KUKA KRL program: MyProgram_185().src

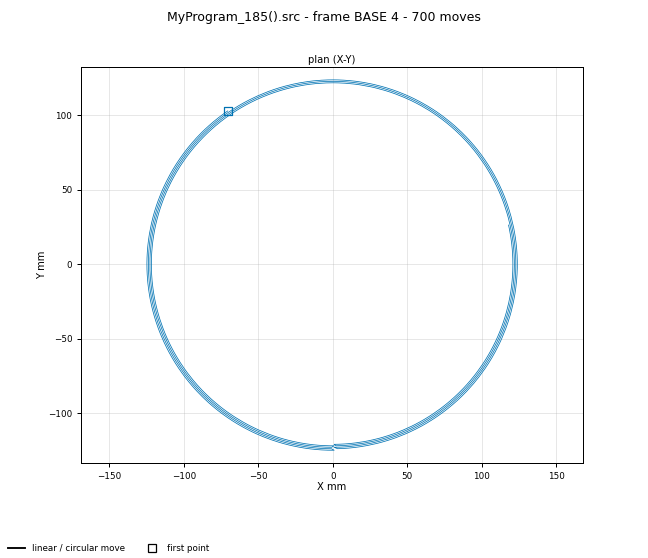
[picture p0: tool path of MyProgram_185().src in frame BASE 4, 700 of 700 moves have a stored position in this frame; points joined in program order, loops and branches not executed]
&ACCESS RVP
&REL 1
&PARAM TEMPLATE = C:\KRC\Roboter\Template\vorgabe
&PARAM EDITMASK = *
DEF MyProgram_185()
; ---- Setting reference (Base) ----
$BASE = BASE_DATA[4]

; --------------------------
; ---- Setting tool (TCP) ----
$TOOL = TOOL_DATA[3]
; --------------------------

$VEL.CP = VEL_APROX_PRINT
Startdeposition()
$VEL.CP = VEL_PRINT
LIN {X -70.5298,Y 102.9618,Z 135,A 120.5149,B 24.9457,C -1.7014,E1 24.9093,E2 685.7205} C_DIS
LIN {X -72.8848,Y 101.309,Z 135,A 122.1964,B 24.9449,C -1.7152,E1 24.9054,E2 684.0005} C_DIS
LIN {X -76.4949,Y 98.6109,Z 135,A 124.23,B 24.9453,C -1.7092,E1 24.9009,E2 681.9739} C_DIS
LIN {X -79.913,Y 95.8627,Z 135,A 126.0592,B 24.9461,C -1.6963,E1 24.897,E2 680.1684} C_DIS
LIN {X -83.1799,Y 93.0413,Z 135,A 128.2007,B 24.9459,C -1.699,E1 24.8925,E2 678.0122} C_DIS
LIN {X -86.1464,Y 90.3016,Z 135,A 130.1225,B 24.9459,C -1.6976,E1 24.8886,E2 676.0856} C_DIS
LIN {X -88.4628,Y 88.0336,Z 135,A 131.6216,B 24.9462,C -1.6945,E1 24.8856,E2 674.5878} C_DIS
LIN {X -91.6049,Y 84.7601,Z 135,A 133.7489,B 24.9464,C -1.6912,E1 24.8815,E2 672.4589} C_DIS
LIN {X -94.5306,Y 81.4834,Z 135,A 135.7394,B 24.9468,C -1.6848,E1 24.8779,E2 670.4747} C_DIS
LIN {X -97.3945,Y 78.0387,Z 135,A 137.8493,B 24.947,C -1.6817,E1 24.8741,E2 668.3623} C_DIS
LIN {X -100.0998,Y 74.5359,Z 135,A 139.8313,B 24.9475,C -1.6739,E1 24.8708,E2 666.3894} C_DIS
LIN {X -102.6203,Y 71.0264,Z 135,A 141.833,B 24.9478,C -1.6692,E1 24.8676,E2 664.3892} C_DIS
LIN {X -104.9174,Y 67.5873,Z 135,A 143.7922,B 24.948,C -1.6665,E1 24.8646,E2 662.4266} C_DIS
LIN {X -107.2782,Y 63.773,Z 135,A 145.689,B 24.9488,C -1.6532,E1 24.8619,E2 660.5516} C_DIS
LIN {X -109.1091,Y 60.5871,Z 135,A 148.347,B 24.9463,C -1.6922,E1 24.8582,E2 657.7868} C_DIS
LIN {X -111.8948,Y 55.2691,Z 135,A 150.3498,B 24.949,C -1.6497,E1 24.8557,E2 655.8745} C_DIS
LIN {X -113.6756,Y 51.5107,Z 135,A 152.2245,B 24.9495,C -1.6423,E1 24.8535,E2 654.0073} C_DIS
LIN {X -115.0996,Y 48.2415,Z 135,A 153.6888,B 24.9502,C -1.6295,E1 24.852,E2 652.5654} C_DIS
LIN {X -116.2639,Y 45.3637,Z 135,A 155.1038,B 24.9505,C -1.6246,E1 24.8505,E2 651.1541} C_DIS
LIN {X -117.2801,Y 42.6692,Z 135,A 156.5898,B 24.9504,C -1.6277,E1 24.8491,E2 649.6522} C_DIS
LIN {X -118.4211,Y 39.3903,Z 135,A 158.1656,B 24.9507,C -1.6219,E1 24.8476,E2 648.0814} C_DIS
LIN {X -119.6405,Y 35.518,Z 135,A 160.0842,B 24.9509,C -1.6184,E1 24.8461,E2 646.16} C_DIS
LIN {X -120.5897,Y 32.1449,Z 135,A 161.5698,B 24.9516,C -1.6077,E1 24.845,E2 644.6913} C_DIS
LIN {X -121.7662,Y 27.3561,Z 135,A 163.8626,B 24.9519,C -1.6016,E1 24.8435,E2 642.3995} C_DIS
LIN {X -123.1315,Y 20.3438,Z 135,A 167.0076,B 24.9529,C -1.5849,E1 24.8419,E2 639.2759} C_DIS
LIN {X -123.7442,Y 16.204,Z 135,A 169.2221,B 24.9525,C -1.5917,E1 24.841,E2 637.032} C_DIS
LIN {X -124.2226,Y 11.9989,Z 135,A 171.157,B 24.9529,C -1.5849,E1 24.8404,E2 635.1015} C_DIS
LIN {X -124.5514,Y 7.8892,Z 135,A 173.0208,B 24.9534,C -1.5774,E1 24.84,E2 633.2444} C_DIS
LIN {X -124.7251,Y 4.3741,Z 135,A 174.7172,B 24.9534,C -1.5757,E1 24.8398,E2 631.5419} C_DIS
LIN {X -124.8019,Y 0.4313,Z 135,A 176.5493,B 24.9538,C -1.5707,E1 24.8398,E2 629.7107} C_DIS
LIN {X -124.7574,Y -3.2955,Z 135,A 178.2564,B 24.9541,C -1.565,E1 24.8398,E2 628.007} C_DIS
LIN {X -124.6055,Y -7.0104,Z 135,A -179.8463,B 24.9539,C -1.5679,E1 24.8402,E2 626.0913} C_DIS
LIN {X -124.202,Y -12.2136,Z 135,A -177.1571,B 24.9536,C -1.5734,E1 24.8409,E2 623.3728} C_DIS
LIN {X -123.7301,Y -16.3119,Z 135,A -175.7455,B 24.9552,C -1.5455,E1 24.8413,E2 622.0193} C_DIS
LIN {X -123.1464,Y -20.2543,Z 135,A -173.8803,B 24.9555,C -1.5413,E1 24.8421,E2 620.1531} C_DIS
LIN {X -122.5805,Y -23.435,Z 135,A -171.8394,B 24.9543,C -1.5618,E1 24.8432,E2 618.0512} C_DIS
LIN {X -121.6545,Y -27.8451,Z 135,A -170.3432,B 24.9562,C -1.5293,E1 24.8441,E2 616.6236} C_DIS
LIN {X -120.7304,Y -31.617,Z 135,A -168.4589,B 24.9562,C -1.5283,E1 24.8454,E2 614.7307} C_DIS
LIN {X -119.8542,Y -34.7881,Z 135,A -167.0168,B 24.9567,C -1.5206,E1 24.8465,E2 613.2987} C_DIS
LIN {X -118.8557,Y -38.0589,Z 135,A -165.4289,B 24.9569,C -1.5165,E1 24.8478,E2 611.7113} C_DIS
LIN {X -117.2331,Y -42.7995,Z 135,A -163.0535,B 24.9571,C -1.513,E1 24.85,E2 609.3308} C_DIS
LIN {X -115.9082,Y -46.2665,Z 135,A -161.3845,B 24.9575,C -1.5063,E1 24.8517,E2 607.6683} C_DIS
LIN {X -114.6553,Y -49.2885,Z 135,A -159.9893,B 24.958,C -1.4971,E1 24.8532,E2 606.2875} C_DIS
LIN {X -113.5275,Y -51.8361,Z 135,A -158.3568,B 24.9573,C -1.5094,E1 24.8551,E2 604.6166} C_DIS
LIN {X -111.3698,Y -56.3204,Z 135,A -156.3247,B 24.9583,C -1.4914,E1 24.8576,E2 602.6164} C_DIS
LIN {X -109.9644,Y -59.0205,Z 135,A -154.8035,B 24.9583,C -1.4931,E1 24.8596,E2 601.083} C_DIS
LIN {X -107.8427,Y -62.8143,Z 135,A -152.8174,B 24.9586,C -1.4872,E1 24.8624,E2 599.1006} C_DIS
LIN {X -105.6364,Y -66.4572,Z 135,A -151.029,B 24.9593,C -1.4744,E1 24.865,E2 597.3336} C_DIS
LIN {X -103.5777,Y -69.6232,Z 135,A -149.0943,B 24.959,C -1.479,E1 24.868,E2 595.3782} C_DIS
LIN {X -101.1976,Y -73.0389,Z 135,A -147.1761,B 24.9593,C -1.4745,E1 24.8711,E2 593.4615} C_DIS
LIN {X -99.0241,Y -75.9595,Z 135,A -145.5031,B 24.9595,C -1.4704,E1 24.8739,E2 591.7901} C_DIS
LIN {X -96.5079,Y -79.1318,Z 135,A -143.63,B 24.9597,C -1.4666,E1 24.8772,E2 589.9174} C_DIS
LIN {X -93.8742,Y -82.2391,Z 135,A -141.7994,B 24.96,C -1.4604,E1 24.8805,E2 588.0933} C_DIS
LIN {X -91.2737,Y -85.1158,Z 135,A -139.9754,B 24.9602,C -1.4584,E1 24.8839,E2 586.2659} C_DIS
LIN {X -87.3757,Y -89.1126,Z 135,A -137.2262,B 24.96,C -1.4615,E1 24.8894,E2 583.4977} C_DIS
LIN {X -83.5883,Y -92.6753,Z 135,A -134.992,B 24.9606,C -1.4494,E1 24.894,E2 581.2832} C_DIS
LIN {X -80.4038,Y -95.4508,Z 135,A -133.0373,B 24.9608,C -1.4464,E1 24.8981,E2 579.3282} C_DIS
LIN {X -76.8747,Y -98.3154,Z 135,A -131.0934,B 24.9614,C -1.4358,E1 24.9023,E2 577.4022} C_DIS
LIN {X -74.1395,Y -100.3942,Z 135,A -129.3572,B 24.9611,C -1.4404,E1 24.9062,E2 575.6488} C_DIS
LIN {X -70.874,Y -102.7256,Z 135,A -127.5006,B 24.9613,C -1.438,E1 24.9105,E2 573.7917} C_DIS
LIN {X -67.2203,Y -105.1523,Z 135,A -125.6255,B 24.9618,C -1.4282,E1 24.9148,E2 571.9335} C_DIS
LIN {X -63.8819,Y -107.2133,Z 135,A -123.7065,B 24.9616,C -1.4311,E1 24.9194,E2 570.0019} C_DIS
LIN {X -60.1893,Y -109.3294,Z 135,A -121.7145,B 24.9616,C -1.4301,E1 24.9243,E2 568.0063} C_DIS
LIN {X -56.8266,Y -111.1121,Z 135,A -120.0688,B 24.9621,C -1.423,E1 24.9283,E2 566.373} C_DIS
LIN {X -53.8577,Y -112.581,Z 135,A -118.5567,B 24.9621,C -1.4208,E1 24.9321,E2 564.8623} C_DIS
LIN {X -50.9392,Y -113.9312,Z 135,A -116.9399,B 24.9619,C -1.4258,E1 24.9363,E2 563.2298} C_DIS
LIN {X -47.0643,Y -115.5866,Z 135,A -115.0807,B 24.9622,C -1.4201,E1 24.941,E2 561.3797} C_DIS
LIN {X -44.084,Y -116.7555,Z 135,A -113.6227,B 24.9623,C -1.4182,E1 24.9448,E2 559.9233} C_DIS
LIN {X -41.333,Y -117.758,Z 135,A -111.5572,B 24.9605,C -1.4517,E1 24.9505,E2 557.7741} C_DIS
LIN {X -36.3107,Y -119.4016,Z 135,A -110.3143,B 24.9637,C -1.393,E1 24.9535,E2 556.6685} C_DIS
LIN {X -33.2824,Y -120.2812,Z 135,A -108.3928,B 24.9625,C -1.4146,E1 24.9588,E2 554.6926} C_DIS
LIN {X -29.5697,Y -121.2473,Z 135,A -106.6724,B 24.9627,C -1.4116,E1 24.9634,E2 552.9768} C_DIS
LIN {X -26.3399,Y -121.9893,Z 135,A -105.1339,B 24.9627,C -1.4116,E1 24.9676,E2 551.4362} C_DIS
LIN {X -22.5131,Y -122.7544,Z 135,A -103.2678,B 24.9625,C -1.4146,E1 24.9727,E2 549.5612} C_DIS
LIN {X -18.5802,Y -123.4109,Z 135,A -101.5071,B 24.9627,C -1.4106,E1 24.9776,E2 547.8082} C_DIS
LIN {X -15.0752,Y -123.8872,Z 135,A -99.847,B 24.9627,C -1.4121,E1 24.9822,E2 546.1434} C_DIS
LIN {X -11.198,Y -124.2993,Z 135,A -97.9834,B 24.9625,C -1.4155,E1 24.9874,E2 544.2708} C_DIS
LIN {X -7.5836,Y -124.5702,Z 135,A -96.3774,B 24.9626,C -1.4127,E1 24.9919,E2 542.6708} C_DIS
LIN {X -3.3227,Y -124.7567,Z 135,A -94.4373,B 24.9626,C -1.4121,E1 24.9973,E2 540.7319} C_DIS
LIN {X 0.8805,Y -124.7969,Z 135,A -92.5835,B 24.9628,C -1.4088,E1 25.0024,E2 538.8859} C_DIS
Enddeposition()
LIN {X 0.8805,Y -124.7969,Z 135,A -92.5835,B 24.9628,C -1.4088,E1 25.0024,E2 538.8859} C_DIS
Startdeposition()
$VEL.CP = VEL_PRINT
LIN {X -0.8634,Y -123.8052,Z 135,A -94.1672,B 24.9639,C -1.3884,E1 24.9979,E2 540.5178} C_DIS
LIN {X -4.5851,Y -123.7233,Z 135,A -95.769,B 24.9636,C -1.3939,E1 24.9934,E2 542.1067} C_DIS
LIN {X -8.0157,Y -123.5489,Z 135,A -97.5065,B 24.964,C -1.3868,E1 24.9885,E2 543.8616} C_DIS
LIN {X -11.6449,Y -123.2592,Z 135,A -99.1179,B 24.9638,C -1.3904,E1 24.9841,E2 545.4653} C_DIS
LIN {X -15.7434,Y -122.8033,Z 135,A -100.884,B 24.9634,C -1.3975,E1 24.9792,E2 547.2159} C_DIS
LIN {X -18.9371,Y -122.351,Z 135,A -102.3711,B 24.9634,C -1.3981,E1 24.9751,E2 548.7027} C_DIS
LIN {X -23.5244,Y -121.5527,Z 135,A -104.6887,B 24.9637,C -1.3911,E1 24.9687,E2 551.0391} C_DIS
LIN {X -27.4993,Y -120.7152,Z 135,A -106.5525,B 24.9637,C -1.3928,E1 24.9636,E2 552.9013} C_DIS
LIN {X -30.9979,Y -119.8657,Z 135,A -108.1238,B 24.9634,C -1.3982,E1 24.9594,E2 554.462} C_DIS
LIN {X -34.2429,Y -118.9794,Z 135,A -109.8275,B 24.9637,C -1.3923,E1 24.9548,E2 556.1823} C_DIS
LIN {X -38.7315,Y -117.5941,Z 135,A -112.0804,B 24.9637,C -1.3903,E1 24.9487,E2 558.444} C_DIS
LIN {X -43.0709,Y -116.0748,Z 135,A -114.0754,B 24.9634,C -1.3984,E1 24.9435,E2 560.4237} C_DIS
LIN {X -46.2408,Y -114.8482,Z 135,A -115.6128,B 24.9632,C -1.4016,E1 24.9395,E2 561.9569} C_DIS
LIN {X -51.3977,Y -112.6365,Z 135,A -118.3361,B 24.9634,C -1.3986,E1 24.9326,E2 564.6939} C_DIS
LIN {X -54.519,Y -111.1578,Z 135,A -119.8207,B 24.963,C -1.4058,E1 24.9288,E2 566.1651} C_DIS
LIN {X -58.9436,Y -108.8787,Z 135,A -122.2823,B 24.9632,C -1.4015,E1 24.9227,E2 568.6436} C_DIS
LIN {X -62.8317,Y -106.6816,Z 135,A -124.1557,B 24.9626,C -1.4134,E1 24.9182,E2 570.4945} C_DIS
LIN {X -67.1902,Y -103.9919,Z 135,A -126.7148,B 24.9628,C -1.4084,E1 24.9121,E2 573.0735} C_DIS
LIN {X -70.8405,Y -101.5402,Z 135,A -128.4781,B 24.962,C -1.4242,E1 24.9081,E2 574.8051} C_DIS
LIN {X -74.3976,Y -98.9637,Z 135,A -130.7859,B 24.9625,C -1.4152,E1 24.9029,E2 577.1426} C_DIS
LIN {X -78.053,Y -96.1074,Z 135,A -132.9335,B 24.9623,C -1.4192,E1 24.8982,E2 579.2887} C_DIS
LIN {X -81.0893,Y -93.5597,Z 135,A -134.8104,B 24.9622,C -1.4208,E1 24.8942,E2 581.169} C_DIS
LIN {X -84.3665,Y -90.6148,Z 135,A -136.7505,B 24.9617,C -1.4295,E1 24.8902,E2 583.0963} C_DIS
LIN {X -87.2827,Y -87.8094,Z 135,A -138.821,B 24.962,C -1.4245,E1 24.886,E2 585.1872} C_DIS
LIN {X -90.5457,Y -84.4407,Z 135,A -140.8885,B 24.9615,C -1.434,E1 24.8821,E2 587.2411} C_DIS
LIN {X -93.5477,Y -81.1033,Z 135,A -143.0184,B 24.9613,C -1.4364,E1 24.8781,E2 589.3748} C_DIS
LIN {X -96.7178,Y -77.2948,Z 135,A -145.1826,B 24.9607,C -1.4477,E1 24.8743,E2 591.5223} C_DIS
LIN {X -99.1413,Y -74.1609,Z 135,A -147.1279,B 24.9607,C -1.4472,E1 24.871,E2 593.478} C_DIS
LIN {X -101.6755,Y -70.646,Z 135,A -149.0677,B 24.9603,C -1.4552,E1 24.8679,E2 595.4081} C_DIS
LIN {X -105.2496,Y -65.2023,Z 135,A -152.17,B 24.9601,C -1.4592,E1 24.8632,E2 598.5166} C_DIS
LIN {X -106.9459,Y -62.3817,Z 135,A -154.0518,B 24.9608,C -1.4475,E1 24.8605,E2 600.4361} C_DIS
LIN {X -108.7995,Y -59.0887,Z 135,A -155.4592,B 24.9597,C -1.4674,E1 24.8587,E2 601.8035} C_DIS
LIN {X -110.4045,Y -56.0283,Z 135,A -156.977,B 24.9592,C -1.4755,E1 24.8567,E2 603.31} C_DIS
LIN {X -111.6365,Y -53.5315,Z 135,A -159.0178,B 24.9608,C -1.4462,E1 24.8542,E2 605.432} C_DIS
LIN {X -113.8153,Y -48.7297,Z 135,A -160.8291,B 24.9589,C -1.4808,E1 24.8523,E2 607.1707} C_DIS
LIN {X -115.2905,Y -45.1275,Z 135,A -163.4083,B 24.9605,C -1.4522,E1 24.8496,E2 609.8326} C_DIS
LIN {X -117.2969,Y -39.6238,Z 135,A -165.323,B 24.9581,C -1.4951,E1 24.8479,E2 611.6559} C_DIS
LIN {X -118.3804,Y -36.255,Z 135,A -166.9438,B 24.9578,C -1.5008,E1 24.8465,E2 613.2723} C_DIS
LIN {X -119.5296,Y -32.267,Z 135,A -168.9037,B 24.9576,C -1.5051,E1 24.845,E2 615.2335} C_DIS
LIN {X -120.3708,Y -28.9693,Z 135,A -170.4394,B 24.9572,C -1.5117,E1 24.844,E2 616.7623} C_DIS
LIN {X -121.1506,Y -25.5205,Z 135,A -172.5728,B 24.9581,C -1.4952,E1 24.8427,E2 618.9478} C_DIS
LIN {X -121.8969,Y -21.669,Z 135,A -174.212,B 24.9574,C -1.5086,E1 24.8419,E2 620.5645} C_DIS
LIN {X -122.5558,Y -17.5632,Z 135,A -175.9083,B 24.9564,C -1.5247,E1 24.8412,E2 622.2325} C_DIS
LIN {X -123.2914,Y -11.3102,Z 135,A -178.6831,B 24.9556,C -1.5402,E1 24.8404,E2 624.9871} C_DIS
LIN {X -123.6607,Y -6.0411,Z 135,A 178.7164,B 24.9555,C -1.5413,E1 24.8399,E2 627.6006} C_DIS
LIN {X -123.7829,Y -2.5424,Z 135,A 176.7623,B 24.956,C -1.5321,E1 24.8398,E2 629.5885} C_DIS
LIN {X -123.806,Y 0.863,Z 135,A 174.9858,B 24.9562,C -1.5286,E1 24.8398,E2 631.3841} C_DIS
LIN {X -123.7022,Y 5.1275,Z 135,A 173.4246,B 24.9548,C -1.553,E1 24.84,E2 632.8965} C_DIS
LIN {X -123.4691,Y 9.1551,Z 135,A 171.6176,B 24.9543,C -1.5617,E1 24.8403,E2 634.6936} C_DIS
LIN {X -123.0248,Y 13.9195,Z 135,A 169.5124,B 24.9536,C -1.5737,E1 24.8409,E2 636.7828} C_DIS
LIN {X -122.5164,Y 17.8392,Z 135,A 167.5366,B 24.9536,C -1.5733,E1 24.8417,E2 638.7713} C_DIS
LIN {X -122.0542,Y 20.7678,Z 135,A 165.467,B 24.9551,C -1.5476,E1 24.8427,E2 640.9144} C_DIS
LIN {X -121.0704,Y 25.8916,Z 135,A 164.0335,B 24.9522,C -1.598,E1 24.8434,E2 642.2364} C_DIS
LIN {X -120.4046,Y 28.8292,Z 135,A 162.2898,B 24.9528,C -1.5872,E1 24.8445,E2 644.016} C_DIS
LIN {X -119.3867,Y 32.7947,Z 135,A 160.4741,B 24.9522,C -1.5967,E1 24.8458,E2 645.8196} C_DIS
LIN {X -118.4389,Y 36.0639,Z 135,A 158.8967,B 24.9519,C -1.6017,E1 24.8471,E2 647.3942} C_DIS
LIN {X -117.4548,Y 39.1499,Z 135,A 157.3941,B 24.9517,C -1.6063,E1 24.8484,E2 648.8945} C_DIS
LIN {X -116.3741,Y 42.2549,Z 135,A 155.7925,B 24.9516,C -1.6076,E1 24.8499,E2 650.502} C_DIS
LIN {X -114.9388,Y 46.0159,Z 135,A 153.9797,B 24.9511,C -1.6156,E1 24.8517,E2 652.3059} C_DIS
LIN {X -113.7774,Y 48.8174,Z 135,A 152.5256,B 24.951,C -1.6177,E1 24.8533,E2 653.763} C_DIS
LIN {X -112.3842,Y 51.9431,Z 135,A 150.9865,B 24.9505,C -1.6246,E1 24.855,E2 655.2943} C_DIS
LIN {X -109.7747,Y 57.2531,Z 135,A 148.3367,B 24.9498,C -1.6367,E1 24.8583,E2 657.9295} C_DIS
LIN {X -106.8363,Y 62.5682,Z 135,A 145.3086,B 24.9498,C -1.6354,E1 24.8625,E2 660.9765} C_DIS
LIN {X -104.6485,Y 66.1623,Z 135,A 143.5116,B 24.9491,C -1.6476,E1 24.8651,E2 662.7536} C_DIS
LIN {X -102.7845,Y 69.0234,Z 135,A 141.7056,B 24.9495,C -1.6422,E1 24.8679,E2 664.5816} C_DIS
LIN {X -100.3296,Y 72.5448,Z 135,A 139.7522,B 24.949,C -1.6492,E1 24.871,E2 666.5279} C_DIS
LIN {X -97.7206,Y 76.0229,Z 135,A 137.7125,B 24.9488,C -1.6534,E1 24.8745,E2 668.5671} C_DIS
LIN {X -95.0962,Y 79.2818,Z 135,A 135.72,B 24.9486,C -1.6561,E1 24.878,E2 670.5625} C_DIS
LIN {X -92.2541,Y 82.5708,Z 135,A 133.7424,B 24.9482,C -1.6628,E1 24.8817,E2 672.533} C_DIS
LIN {X -89.2417,Y 85.8185,Z 135,A 131.6496,B 24.948,C -1.6661,E1 24.8857,E2 674.6271} C_DIS
LIN {X -86.2463,Y 88.8277,Z 135,A 129.8454,B 24.9472,C -1.678,E1 24.8892,E2 676.4106} C_DIS
LIN {X -84.2676,Y 90.7069,Z 135,A 128.4959,B 24.9472,C -1.6772,E1 24.892,E2 677.7675} C_DIS
LIN {X -81.9548,Y 92.8018,Z 135,A 126.9872,B 24.9472,C -1.6777,E1 24.8951,E2 679.2811} C_DIS
LIN {X -78.6554,Y 95.6151,Z 135,A 124.9342,B 24.9471,C -1.6802,E1 24.8995,E2 681.3361} C_DIS
LIN {X -74.843,Y 98.6276,Z 135,A 122.5516,B 24.9471,C -1.6791,E1 24.9048,E2 683.73} C_DIS
LIN {X -70.7218,Y 101.6227,Z 135,A 120.3716,B 24.9464,C -1.6919,E1 24.9097,E2 685.8871} C_DIS
LIN {X -67.0782,Y 104.0645,Z 135,A 118.2542,B 24.9464,C -1.6919,E1 24.9147,E2 688.0113} C_DIS
LIN {X -63.1803,Y 106.4756,Z 135,A 116.1758,B 24.946,C -1.6978,E1 24.9196,E2 690.0821} C_DIS
LIN {X -59.6094,Y 108.5155,Z 135,A 114.2639,B 24.9458,C -1.7008,E1 24.9243,E2 691.9925} C_DIS
LIN {X -56.1238,Y 110.3559,Z 135,A 111.5295,B 24.9482,C -1.6632,E1 24.9314,E2 694.8236} C_DIS
LIN {X -50.3029,Y 113.1283,Z 135,A 109.6719,B 24.9447,C -1.7183,E1 24.9357,E2 696.5549} C_DIS
LIN {X -43.599,Y 115.877,Z 135,A 106.0494,B 24.9452,C -1.7107,E1 24.9452,E2 700.2034} C_DIS
LIN {X -39.3794,Y 117.3783,Z 135,A 104.085,B 24.9447,C -1.7182,E1 24.9503,E2 702.1536} C_DIS
LIN {X -36.2539,Y 118.3807,Z 135,A 102.0224,B 24.9461,C -1.6953,E1 24.956,E2 704.2743} C_DIS
LIN {X -32.1251,Y 119.5675,Z 135,A 100.4225,B 24.9449,C -1.715,E1 24.9602,E2 705.8299} C_DIS
LIN {X -26.7788,Y 120.8779,Z 135,A 97.401,B 24.9461,C -1.6958,E1 24.9685,E2 708.901} C_DIS
LIN {X -22.2265,Y 121.7971,Z 135,A 96.0414,B 24.9437,C -1.7337,E1 24.972,E2 710.172} C_DIS
LIN {X -16.735,Y 122.6734,Z 135,A 93.1682,B 24.9445,C -1.7215,E1 24.98,E2 713.0765} C_DIS
LIN {X -12.7982,Y 123.1455,Z 135,A 91.3595,B 24.9443,C -1.7238,E1 24.985,E2 714.881} C_DIS
LIN {X -7.7164,Y 123.5673,Z 135,A 88.8747,B 24.9446,C -1.7191,E1 24.992,E2 717.3781} C_DIS
LIN {X -3.327,Y 123.7634,Z 135,A 87.0723,B 24.9439,C -1.7304,E1 24.9969,E2 719.1539} C_DIS
LIN {X 0.4786,Y 123.8073,Z 135,A 85.3464,B 24.9438,C -1.7324,E1 25.0018,E2 720.875} C_DIS
LIN {X 3.4843,Y 123.759,Z 135,A 83.9026,B 24.9438,C -1.7302,E1 25.0058,E2 722.324} C_DIS
LIN {X 7.3163,Y 123.592,Z 135,A 82.0806,B 24.944,C -1.728,E1 25.0109,E2 724.1504} C_DIS
LIN {X 11.2885,Y 123.2934,Z 135,A 80.3604,B 24.9437,C -1.7337,E1 25.0156,E2 725.8563} C_DIS
LIN {X 15.3492,Y 122.8547,Z 135,A 78.4456,B 24.9437,C -1.7321,E1 25.021,E2 727.7733} C_DIS
LIN {X 20.4607,Y 122.1055,Z 135,A 75.9717,B 24.9441,C -1.7275,E1 25.0278,E2 730.2558} C_DIS
LIN {X 25.2617,Y 121.2046,Z 135,A 73.7833,B 24.9439,C -1.7299,E1 25.0338,E2 732.436} C_DIS
LIN {X 27.8274,Y 120.6402,Z 135,A 72.2715,B 24.9449,C -1.7153,E1 25.038,E2 733.9804} C_DIS
LIN {X 32.6518,Y 119.4267,Z 135,A 70.2825,B 24.944,C -1.7287,E1 25.0433,E2 735.9347} C_DIS
LIN {X 35.9969,Y 118.4594,Z 135,A 68.444,B 24.9448,C -1.7167,E1 25.0483,E2 737.7983} C_DIS
LIN {X 40.359,Y 117.045,Z 135,A 66.4923,B 24.9444,C -1.723,E1 25.0534,E2 739.7313} C_DIS
LIN {X 43.5983,Y 115.8773,Z 135,A 64.9987,B 24.9441,C -1.7263,E1 25.0573,E2 741.2139} C_DIS
LIN {X 48.3745,Y 113.9681,Z 135,A 62.428,B 24.9449,C -1.7146,E1 25.064,E2 743.8064} C_DIS
LIN {X 51.7715,Y 112.4636,Z 135,A 60.8091,B 24.9447,C -1.7174,E1 25.0681,E2 745.4146} C_DIS
LIN {X 54.4905,Y 111.1719,Z 135,A 59.2781,B 24.9453,C -1.709,E1 25.0719,E2 746.9614} C_DIS
LIN {X 58.7828,Y 108.9651,Z 135,A 57.165,B 24.9451,C -1.7118,E1 25.0771,E2 749.062} C_DIS
LIN {X 63.3289,Y 106.3871,Z 135,A 54.7431,B 24.9453,C -1.7081,E1 25.083,E2 751.4853} C_DIS
LIN {X 66.9379,Y 104.1543,Z 135,A 52.7664,B 24.9456,C -1.7044,E1 25.0877,E2 753.4645} C_DIS
LIN {X 69.8659,Y 102.2133,Z 135,A 51.1048,B 24.9458,C -1.6999,E1 25.0915,E2 755.1311} C_DIS
LIN {X 73.5379,Y 99.6043,Z 135,A 49.0505,B 24.946,C -1.6977,E1 25.0962,E2 757.1833} C_DIS
LIN {X 76.8628,Y 97.0616,Z 135,A 47.3226,B 24.9456,C -1.7044,E1 25.0999,E2 758.8891} C_DIS
LIN {X 78.8901,Y 95.4208,Z 135,A 45.8834,B 24.9464,C -1.6907,E1 25.1031,E2 760.3553} C_DIS
LIN {X 81.6527,Y 93.0683,Z 135,A 44.0653,B 24.9471,C -1.6805,E1 25.107,E2 762.1903} C_DIS
LIN {X 86.4832,Y 88.5974,Z 135,A 41.1856,B 24.947,C -1.6823,E1 25.1128,E2 765.0539} C_DIS
LIN {X 89.6786,Y 85.3614,Z 135,A 39.2614,B 24.9467,C -1.6865,E1 25.1165,E2 766.9598} C_DIS
LIN {X 91.9511,Y 82.908,Z 135,A 37.5683,B 24.9474,C -1.6758,E1 25.1197,E2 768.6707} C_DIS
LIN {X 94.7944,Y 79.6416,Z 135,A 35.2848,B 24.9485,C -1.6573,E1 25.1239,E2 770.9877} C_DIS
LIN {X 97.0694,Y 76.853,Z 135,A 33.9235,B 24.9478,C -1.6682,E1 25.1262,E2 772.3167} C_DIS
LIN {X 99.6033,Y 73.5393,Z 135,A 32.3056,B 24.9472,C -1.679,E1 25.1289,E2 773.9015} C_DIS
LIN {X 101.9529,Y 70.2454,Z 135,A 30.1541,B 24.9483,C -1.6603,E1 25.1324,E2 776.0867} C_DIS
LIN {X 104.2542,Y 66.7818,Z 135,A 28.2901,B 24.9485,C -1.6582,E1 25.1353,E2 777.9461} C_DIS
LIN {X 106.2415,Y 63.5732,Z 135,A 26.4971,B 24.9489,C -1.6512,E1 25.1379,E2 779.7467} C_DIS
LIN {X 108.3313,Y 59.9424,Z 135,A 24.6332,B 24.949,C -1.6496,E1 25.1404,E2 781.6046} C_DIS
LIN {X 110.1536,Y 56.5211,Z 135,A 23.0598,B 24.9486,C -1.6557,E1 25.1424,E2 783.1554} C_DIS
LIN {X 112.0075,Y 52.7536,Z 135,A 20.7114,B 24.9502,C -1.6297,E1 25.1454,E2 785.5524} C_DIS
LIN {X 114.0055,Y 48.285,Z 135,A 18.6368,B 24.9501,C -1.6326,E1 25.1477,E2 787.6087} C_DIS
LIN {X 115.3485,Y 44.9785,Z 135,A 17.0089,B 24.9503,C -1.629,E1 25.1493,E2 789.2363} C_DIS
LIN {X 116.7642,Y 41.1689,Z 135,A 15.12,B 24.9507,C -1.6228,E1 25.1511,E2 791.129} C_DIS
LIN {X 118.041,Y 37.3468,Z 135,A 12.5227,B 24.9532,C -1.5804,E1 25.1534,E2 793.8116} C_DIS
LIN {X 119.6003,Y 32.0018,Z 135,A 10.7795,B 24.9512,C -1.6143,E1 25.1546,E2 795.4651} C_DIS
LIN {X 121.422,Y 24.1935,Z 135,A 6.7226,B 24.9529,C -1.585,E1 25.1571,E2 799.5673} C_DIS
LIN {X 122.044,Y 20.8292,Z 135,A 5.5154,B 24.9521,C -1.599,E1 25.1577,E2 800.7345} C_DIS
LIN {X 122.5743,Y 17.4338,Z 135,A 4.0226,B 24.9521,C -1.5988,E1 25.1583,E2 802.2189} C_DIS
LIN {X 123.0399,Y 13.7795,Z 135,A 2.1577,B 24.9529,C -1.5851,E1 25.1589,E2 804.105} C_DIS
LIN {X 123.3983,Y 10.0698,Z 135,A 0.4241,B 24.9533,C -1.5791,E1 25.1594,E2 805.8425} C_DIS
LIN {X 123.6575,Y 6.1039,Z 135,A -1.3708,B 24.9535,C -1.5753,E1 25.1596,E2 807.6357} C_DIS
LIN {X 123.7885,Y 2.2028,Z 135,A -3.1251,B 24.9537,C -1.5721,E1 25.1598,E2 809.3873} C_DIS
LIN {X 123.7873,Y -2.2781,Z 135,A -5.2586,B 24.9543,C -1.5622,E1 25.1598,E2 811.5313} C_DIS
LIN {X 123.6329,Y -6.5938,Z 135,A -7.2503,B 24.9546,C -1.556,E1 25.1595,E2 813.5258} C_DIS
LIN {X 123.3609,Y -10.5126,Z 135,A -8.8072,B 24.9542,C -1.5633,E1 25.1592,E2 815.0562} C_DIS
LIN {X 122.7356,Y -16.2602,Z 135,A -11.637,B 24.9552,C -1.5466,E1 25.1583,E2 817.9086} C_DIS
LIN {X 122.137,Y -20.2718,Z 135,A -13.3908,B 24.9552,C -1.5467,E1 25.1575,E2 819.6518} C_DIS
LIN {X 121.1872,Y -25.3473,Z 135,A -15.7969,B 24.9557,C -1.5381,E1 25.1562,E2 822.0643} C_DIS
LIN {X 119.6616,Y -31.772,Z 135,A -18.8752,B 24.9563,C -1.527,E1 25.1542,E2 825.1509} C_DIS
LIN {X 118.9726,Y -34.2661,Z 135,A -20.7014,B 24.9583,C -1.4913,E1 25.1527,E2 827.0508} C_DIS
LIN {X 117.5762,Y -38.7851,Z 135,A -22.3644,B 24.9572,C -1.5109,E1 25.1513,E2 828.6582} C_DIS
LIN {X 116.0865,Y -43.0396,Z 135,A -24.3489,B 24.9573,C -1.5094,E1 25.1495,E2 830.635} C_DIS
LIN {X 113.1249,Y -50.3104,Z 135,A -27.9212,B 24.9578,C -1.5012,E1 25.1456,E2 834.2071} C_DIS
LIN {X 111.7493,Y -53.2953,Z 135,A -29.3847,B 24.9578,C -1.4994,E1 25.1439,E2 835.6668} C_DIS
LIN {X 110.4143,Y -56.0091,Z 135,A -30.5836,B 24.9575,C -1.5054,E1 25.1424,E2 836.8452} C_DIS
LIN {X 109.1597,Y -58.4206,Z 135,A -32.2707,B 24.959,C -1.4798,E1 25.1402,E2 838.5838} C_DIS
LIN {X 106.8285,Y -62.5816,Z 135,A -34.3576,B 24.959,C -1.4793,E1 25.1373,E2 840.661} C_DIS
LIN {X 104.4943,Y -66.4066,Z 135,A -36.4435,B 24.9594,C -1.4727,E1 25.1342,E2 842.752} C_DIS
LIN {X 102.1347,Y -69.9805,Z 135,A -38.3957,B 24.9596,C -1.4685,E1 25.1312,E2 844.7043} C_DIS
LIN {X 98.2445,Y -75.3445,Z 135,A -42.2266,B 24.9621,C -1.4218,E1 25.1246,E2 848.6271} C_DIS
LIN {X 94.5111,Y -79.9779,Z 135,A -43.977,B 24.9598,C -1.4646,E1 25.1217,E2 850.2684} C_DIS
LIN {X 89.6786,Y -85.3614,Z 135,A -47.9999,B 24.9621,C -1.4222,E1 25.1139,E2 854.3738} C_DIS
LIN {X 86.501,Y -88.5799,Z 135,A -49.574,B 24.961,C -1.4429,E1 25.1109,E2 855.8923} C_DIS
LIN {X 83.9624,Y -90.9897,Z 135,A -51.5909,B 24.9623,C -1.4192,E1 25.1067,E2 857.9571} C_DIS
LIN {X 80.9625,Y -93.669,Z 135,A -53.6152,B 24.9629,C -1.4068,E1 25.1023,E2 860.0026} C_DIS
LIN {X 77.2318,Y -96.7679,Z 135,A -55.2948,B 24.9617,C -1.4298,E1 25.0988,E2 861.6216} C_DIS
LIN {X 74.7202,Y -98.7202,Z 135,A -56.8709,B 24.9622,C -1.4214,E1 25.0953,E2 863.2117} C_DIS
LIN {X 71.8821,Y -100.8055,Z 135,A -58.8153,B 24.9632,C -1.4024,E1 25.0908,E2 865.1943} C_DIS
LIN {X 68.3507,Y -103.233,Z 135,A -60.3822,B 24.9623,C -1.419,E1 25.0873,E2 866.7168} C_DIS
LIN {X 65.7863,Y -104.8859,Z 135,A -62.0499,B 24.9631,C -1.4036,E1 25.0833,E2 868.4155} C_DIS
LIN {X 62.7803,Y -106.7116,Z 135,A -63.6731,B 24.9632,C -1.4007,E1 25.0793,E2 870.0404} C_DIS
LIN {X 59.633,Y -108.5026,Z 135,A -65.0729,B 24.9627,C -1.4113,E1 25.076,E2 871.4111} C_DIS
LIN {X 55.6358,Y -110.6043,Z 135,A -67.6081,B 24.964,C -1.3859,E1 25.0696,E2 873.9994} C_DIS
LIN {X 51.6734,Y -112.509,Z 135,A -69.097,B 24.9628,C -1.4095,E1 25.0659,E2 875.4289} C_DIS
LIN {X 48.2515,Y -114.0195,Z 135,A -70.8057,B 24.9628,C -1.4079,E1 25.0615,E2 877.1372} C_DIS
LIN {X 45.0355,Y -115.3263,Z 135,A -72.3854,B 24.9629,C -1.4069,E1 25.0575,E2 878.7155} C_DIS
LIN {X 42.4678,Y -116.2973,Z 135,A -73.7162,B 24.9632,C -1.4022,E1 25.0539,E2 880.0547} C_DIS
LIN {X 39.4705,Y -117.348,Z 135,A -75.1609,B 24.9632,C -1.4016,E1 25.0501,E2 881.4981} C_DIS
LIN {X 36.5458,Y -118.2914,Z 135,A -76.9005,B 24.9641,C -1.3844,E1 25.0454,E2 883.2752} C_DIS
LIN {X 33.2908,Y -119.2479,Z 135,A -78.093,B 24.9632,C -1.401,E1 25.0423,E2 884.4263} C_DIS
LIN {X 29.6391,Y -120.2094,Z 135,A -79.9692,B 24.9637,C -1.3929,E1 25.0372,E2 886.3189} C_DIS
LIN {X 25.9768,Y -121.052,Z 135,A -81.5902,B 24.9634,C -1.3971,E1 25.0328,E2 887.928} C_DIS
LIN {X 23.1981,Y -121.6151,Z 135,A -83.4718,B 24.9649,C -1.3684,E1 25.0275,E2 889.8751} C_DIS
LIN {X 18.797,Y -122.3727,Z 135,A -84.7939,B 24.9631,C -1.4028,E1 25.0241,E2 891.1145} C_DIS
LIN {X 14.4604,Y -122.9607,Z 135,A -87.0641,B 24.9638,C -1.3896,E1 25.0177,E2 893.4141} C_DIS
LIN {X 10.3711,Y -123.3728,Z 135,A -88.868,B 24.9636,C -1.3933,E1 25.0127,E2 895.2082} C_DIS
LIN {X 7.3879,Y -123.5876,Z 135,A -90.3682,B 24.964,C -1.3871,E1 25.0085,E2 896.7225} C_DIS
LIN {X 3.203,Y -123.7668,Z 135,A -92.3139,B 24.964,C -1.3861,E1 25.003,E2 898.6701} C_DIS
LIN {X 3.203,Y -123.7668,Z 135,A -92.3139,B 24.964,C -1.3861,E1 25.003,E2 898.6701} C_DIS
Enddeposition()
LIN {X 0.8675,Y -122.8108,Z 135,A -92.672,B 24.9613,C -1.4379,E1 25.0024,E2 898.9054} C_DIS
Startdeposition()
$VEL.CP = VEL_PRINT
LIN {X 4.7527,Y -122.7233,Z 135,A -90.739,B 24.9609,C -1.4443,E1 25.0078,E2 896.9577} C_DIS
LIN {X 8.1451,Y -122.5461,Z 135,A -89.1619,B 24.9609,C -1.4445,E1 25.0122,E2 895.3806} C_DIS
LIN {X 11.6911,Y -122.2574,Z 135,A -87.5647,B 24.961,C -1.4424,E1 25.0166,E2 893.7894} C_DIS
LIN {X 18.944,Y -121.3453,Z 135,A -84.5708,B 24.962,C -1.4244,E1 25.0248,E2 890.8404} C_DIS
LIN {X 25.8677,Y -120.0599,Z 135,A -80.9369,B 24.9609,C -1.4439,E1 25.0349,E2 887.1646} C_DIS
LIN {X 30.969,Y -118.8478,Z 135,A -78.5477,B 24.9609,C -1.4436,E1 25.0414,E2 884.7797} C_DIS
LIN {X 36.4645,Y -117.278,Z 135,A -75.6886,B 24.9603,C -1.456,E1 25.0491,E2 881.896} C_DIS
LIN {X 40.0763,Y -116.0922,Z 135,A -74.0159,B 24.9604,C -1.4533,E1 25.0535,E2 880.233} C_DIS
LIN {X 42.5353,Y -115.2153,Z 135,A -72.5513,B 24.9597,C -1.4671,E1 25.0574,E2 878.7388} C_DIS
LIN {X 47.0709,Y -113.4367,Z 135,A -70.5099,B 24.9601,C -1.459,E1 25.0626,E2 876.7213} C_DIS
LIN {X 49.7814,Y -112.2739,Z 135,A -68.6482,B 24.9587,C -1.4852,E1 25.0675,E2 874.8021} C_DIS
LIN {X 53.5488,Y -110.5277,Z 135,A -67.2666,B 24.96,C -1.4607,E1 25.0708,E2 873.4821} C_DIS
LIN {X 56.7041,Y -108.9417,Z 135,A -65.5283,B 24.9596,C -1.468,E1 25.0752,E2 871.7313} C_DIS
LIN {X 60.1697,Y -107.0678,Z 135,A -63.0968,B 24.9578,C -1.501,E1 25.0813,E2 869.2289} C_DIS
LIN {X 64.3173,Y -104.6289,Z 135,A -61.445,B 24.9592,C -1.4755,E1 25.0851,E2 867.6425} C_DIS
LIN {X 67.9003,Y -102.3405,Z 135,A -59.4115,B 24.9589,C -1.482,E1 25.0899,E2 865.6006} C_DIS
LIN {X 72.0212,Y -99.483,Z 135,A -56.6063,B 24.9573,C -1.5103,E1 25.0964,E2 862.738} C_DIS
LIN {X 75.6827,Y -96.7269,Z 135,A -55.0007,B 24.9585,C -1.4881,E1 25.0998,E2 861.1908} C_DIS
LIN {X 80.4985,Y -92.7578,Z 135,A -52.3945,B 24.959,C -1.4794,E1 25.1053,E2 858.6153} C_DIS
LIN {X 85.1401,Y -88.5169,Z 135,A -49.4514,B 24.9586,C -1.4868,E1 25.1114,E2 855.6665} C_DIS
LIN {X 89.125,Y -84.5028,Z 135,A -46.8035,B 24.9582,C -1.4938,E1 25.1166,E2 853.0135} C_DIS
LIN {X 93.0824,Y -80.1223,Z 135,A -43.8386,B 24.9572,C -1.5116,E1 25.1221,E2 850.0199} C_DIS
LIN {X 95.0247,Y -77.8089,Z 135,A -41.8263,B 24.9552,C -1.5461,E1 25.1258,E2 847.9355} C_DIS
LIN {X 98.0584,Y -73.9491,Z 135,A -39.9136,B 24.956,C -1.5331,E1 25.129,E2 846.0626} C_DIS
LIN {X 100.9341,Y -69.9733,Z 135,A -37.9436,B 24.9565,C -1.5233,E1 25.1321,E2 844.1253} C_DIS
LIN {X 103.1186,Y -66.712,Z 135,A -36.0366,B 24.956,C -1.5324,E1 25.135,E2 842.2064} C_DIS
LIN {X 105.3249,Y -63.172,Z 135,A -34.1313,B 24.9558,C -1.536,E1 25.1378,E2 840.3023} C_DIS
LIN {X 107.6252,Y -59.1681,Z 135,A -31.5585,B 24.9542,C -1.5638,E1 25.1414,E2 837.6772} C_DIS
LIN {X 109.4445,Y -55.7257,Z 135,A -30.0234,B 24.9547,C -1.5549,E1 25.1433,E2 836.1712} C_DIS
LIN {X 111.2415,Y -52.049,Z 135,A -28.0318,B 24.9541,C -1.565,E1 25.1457,E2 834.1667} C_DIS
LIN {X 114.4385,Y -44.5793,Z 135,A -24.5744,B 24.9544,C -1.5597,E1 25.1494,E2 830.7408} C_DIS
LIN {X 115.6095,Y -41.4483,Z 135,A -23.0132,B 24.9541,C -1.5647,E1 25.1509,E2 829.1765} C_DIS
LIN {X 116.4143,Y -39.1322,Z 135,A -20.8969,B 24.9509,C -1.6185,E1 25.1528,E2 826.9454} C_DIS
LIN {X 118.3161,Y -32.9369,Z 135,A -18.8804,B 24.9535,C -1.5762,E1 25.1543,E2 825.0401} C_DIS
LIN {X 119.4205,Y -28.6751,Z 135,A -16.5156,B 24.9521,C -1.5988,E1 25.1559,E2 822.6357} C_DIS
LIN {X 120.1711,Y -25.3527,Z 135,A -14.513,B 24.9505,C -1.6253,E1 25.1571,E2 820.5823} C_DIS
LIN {X 121.1504,Y -20.1528,Z 135,A -12.8026,B 24.9524,C -1.5943,E1 25.1578,E2 818.9549} C_DIS
LIN {X 121.5955,Y -17.2657,Z 135,A -10.8946,B 24.9504,C -1.6268,E1 25.1586,E2 816.9816} C_DIS
LIN {X 122.1442,Y -12.8238,Z 135,A -9.4514,B 24.952,C -1.6005,E1 25.159,E2 815.6089} C_DIS
LIN {X 122.4711,Y -9.1905,Z 135,A -7.6917,B 24.9515,C -1.6091,E1 25.1594,E2 813.8394} C_DIS
LIN {X 122.6932,Y -5.5126,Z 135,A -5.8979,B 24.9509,C -1.6186,E1 25.1597,E2 812.034} C_DIS
LIN {X 122.8025,Y -1.7892,Z 135,A -4.2353,B 24.9508,C -1.6204,E1 25.1597,E2 810.3768} C_DIS
LIN {X 122.7919,Y 2.4282,Z 135,A -2.2106,B 24.9502,C -1.6298,E1 25.1597,E2 808.3421} C_DIS
LIN {X 122.6502,Y 6.3676,Z 135,A -0.4125,B 24.95,C -1.6337,E1 25.1595,E2 806.5455} C_DIS
LIN {X 122.372,Y 10.4246,Z 135,A 1.4346,B 24.9498,C -1.6374,E1 25.1591,E2 804.7008} C_DIS
LIN {X 121.9672,Y 14.4077,Z 135,A 3.1074,B 24.95,C -1.6335,E1 25.1586,E2 803.047} C_DIS
LIN {X 121.4635,Y 18.181,Z 135,A 5.0943,B 24.949,C -1.6499,E1 25.1578,E2 801.0331} C_DIS
LIN {X 120.2751,Y 24.851,Z 135,A 8.3742,B 24.948,C -1.6661,E1 25.1561,E2 797.7343} C_DIS
LIN {X 118.9114,Y 30.7223,Z 135,A 11.0098,B 24.948,C -1.6659,E1 25.1544,E2 795.1144} C_DIS
LIN {X 117.0338,Y 37.2372,Z 135,A 14.062,B 24.9477,C -1.67,E1 25.152,E2 792.0699} C_DIS
LIN {X 116.0091,Y 40.3159,Z 135,A 15.5668,B 24.9475,C -1.6741,E1 25.1506,E2 790.5638} C_DIS
LIN {X 114.7742,Y 43.7131,Z 135,A 17.3686,B 24.9468,C -1.685,E1 25.1488,E2 788.7465} C_DIS
LIN {X 113.3264,Y 47.3348,Z 135,A 19.0698,B 24.9468,C -1.6844,E1 25.1471,E2 787.056} C_DIS
LIN {X 111.8907,Y 50.6381,Z 135,A 21.0709,B 24.9455,C -1.7056,E1 25.1447,E2 785.0159} C_DIS
LIN {X 110.4753,Y 53.6584,Z 135,A 22.4058,B 24.9459,C -1.6988,E1 25.1431,E2 783.7042} C_DIS
LIN {X 108.9193,Y 56.7468,Z 135,A 23.9094,B 24.9459,C -1.6978,E1 25.1412,E2 782.2108} C_DIS
LIN {X 107.15,Y 60.0234,Z 135,A 25.6321,B 24.9457,C -1.7019,E1 25.1389,E2 780.4876} C_DIS
LIN {X 105.2317,Y 63.3267,Z 135,A 27.504,B 24.9451,C -1.7113,E1 25.1362,E2 778.6032} C_DIS
LIN {X 102.8558,Y 67.1169,Z 135,A 29.4716,B 24.9451,C -1.7108,E1 25.1333,E2 776.6466} C_DIS
LIN {X 100.1837,Y 71.0438,Z 135,A 31.7947,B 24.9444,C -1.7219,E1 25.1296,E2 774.3086} C_DIS
LIN {X 97.6472,Y 74.4913,Z 135,A 33.7486,B 24.9443,C -1.7247,E1 25.1263,E2 772.3573} C_DIS
LIN {X 95.6489,Y 77.0402,Z 135,A 35.5771,B 24.943,C -1.7443,E1 25.123,E2 770.4911} C_DIS
LIN {X 93.2806,Y 79.8922,Z 135,A 36.9908,B 24.9437,C -1.7326,E1 25.1205,E2 769.1116} C_DIS
LIN {X 90.6537,Y 82.8609,Z 135,A 38.9148,B 24.9432,C -1.7406,E1 25.1169,E2 767.1773} C_DIS
LIN {X 87.4534,Y 86.2318,Z 135,A 40.985,B 24.9432,C -1.7405,E1 25.1129,E2 765.1163} C_DIS
LIN {X 85.3462,Y 88.3173,Z 135,A 42.852,B 24.9414,C -1.7676,E1 25.1091,E2 763.1931} C_DIS
LIN {X 82.029,Y 91.4066,Z 135,A 44.4487,B 24.9429,C -1.7461,E1 25.1059,E2 761.6535} C_DIS
LIN {X 78.7209,Y 94.271,Z 135,A 46.6389,B 24.9421,C -1.7575,E1 25.1012,E2 759.4449} C_DIS
LIN {X 74.8849,Y 97.3462,Z 135,A 48.8105,B 24.9422,C -1.7557,E1 25.0964,E2 757.2855} C_DIS
LIN {X 71.3881,Y 99.9382,Z 135,A 50.8059,B 24.9422,C -1.7576,E1 25.0919,E2 755.2928} C_DIS
LIN {X 68.6072,Y 101.8676,Z 135,A 52.4047,B 24.9419,C -1.7612,E1 25.0882,E2 753.6908} C_DIS
LIN {X 64.993,Y 104.2105,Z 135,A 54.1505,B 24.9425,C -1.7515,E1 25.0842,E2 751.9736} C_DIS
LIN {X 61.8307,Y 106.1171,Z 135,A 56.1723,B 24.9414,C -1.7687,E1 25.0792,E2 749.9174} C_DIS
LIN {X 57.7687,Y 108.3827,Z 135,A 58.2174,B 24.9416,C -1.7656,E1 25.0742,E2 747.8855} C_DIS
LIN {X 54.8624,Y 109.8814,Z 135,A 59.7516,B 24.9414,C -1.768,E1 25.0704,E2 746.3497} C_DIS
LIN {X 50.9535,Y 111.7481,Z 135,A 61.8241,B 24.9411,C -1.773,E1 25.0652,E2 744.2708} C_DIS
LIN {X 45.6905,Y 113.9996,Z 135,A 64.6113,B 24.9405,C -1.7815,E1 25.0579,E2 741.4699} C_DIS
LIN {X 41.4745,Y 115.6001,Z 135,A 66.4816,B 24.9411,C -1.7722,E1 25.0531,E2 739.6255} C_DIS
LIN {X 37.7954,Y 116.8555,Z 135,A 68.6066,B 24.94,C -1.7887,E1 25.0474,E2 737.4654} C_DIS
LIN {X 34.7041,Y 117.8099,Z 135,A 69.7813,B 24.941,C -1.7738,E1 25.0443,E2 736.3282} C_DIS
LIN {X 31.6577,Y 118.6647,Z 135,A 71.3115,B 24.9408,C -1.7774,E1 25.0402,E2 734.792} C_DIS
LIN {X 27.6018,Y 119.6734,Z 135,A 73.2943,B 24.9406,C -1.78,E1 25.0348,E2 732.8057} C_DIS
LIN {X 20.9466,Y 121.0176,Z 135,A 77.171,B 24.9382,C -1.8153,E1 25.0239,E2 728.8498} C_DIS
LIN {X 15.5318,Y 121.8298,Z 135,A 78.8015,B 24.9412,C -1.7718,E1 25.0197,E2 727.3236} C_DIS
LIN {X 12.5793,Y 122.1705,Z 135,A 80.392,B 24.9405,C -1.7817,E1 25.0152,E2 725.7109} C_DIS
LIN {X 8.6968,Y 122.5071,Z 135,A 82.2065,B 24.9405,C -1.7817,E1 25.0102,E2 723.8974} C_DIS
LIN {X 4.739,Y 122.7238,Z 135,A 83.9882,B 24.9407,C -1.7784,E1 25.0052,E2 722.124} C_DIS
LIN {X 0.838,Y 122.8125,Z 135,A 85.8366,B 24.9407,C -1.7794,E1 25.0001,E2 720.2733} C_DIS
LIN {X -3.2439,Y 122.7725,Z 135,A 87.6589,B 24.9409,C -1.7751,E1 24.995,E2 718.4612} C_DIS
LIN {X -8.7463,Y 122.5035,Z 135,A 90.2725,B 24.9409,C -1.7762,E1 24.9877,E2 715.8443} C_DIS
LIN {X -15.3027,Y 121.8598,Z 135,A 93.2728,B 24.9412,C -1.771,E1 24.9794,E2 712.8544} C_DIS
LIN {X -18.9666,Y 121.3418,Z 135,A 95.5794,B 24.9395,C -1.7969,E1 24.9729,E2 710.4845} C_DIS
LIN {X -22.9732,Y 120.6473,Z 135,A 96.6612,B 24.9421,C -1.7576,E1 24.9702,E2 709.4948} C_DIS
LIN {X -28.7488,Y 119.4028,Z 135,A 99.76,B 24.9412,C -1.7708,E1 24.9616,E2 706.3607} C_DIS
LIN {X -32.5387,Y 118.4274,Z 135,A 101.7187,B 24.9409,C -1.775,E1 24.9563,E2 704.3891} C_DIS
LIN {X -36.9289,Y 117.1323,Z 135,A 103.7602,B 24.9414,C -1.7683,E1 24.9509,E2 702.3601} C_DIS
LIN {X -40.111,Y 116.0802,Z 135,A 105.2485,B 24.9418,C -1.7629,E1 24.947,E2 700.8817} C_DIS
LIN {X -42.6194,Y 115.1838,Z 135,A 107.4877,B 24.9388,C -1.8071,E1 24.9409,E2 698.5328} C_DIS
LIN {X -48.4198,Y 112.8677,Z 135,A 109.4621,B 24.942,C -1.7597,E1 24.936,E2 696.6667} C_DIS
LIN {X -51.6281,Y 111.4361,Z 135,A 110.8416,B 24.9429,C -1.7454,E1 24.9326,E2 695.3178} C_DIS
LIN {X -55.7333,Y 109.4406,Z 135,A 113.3424,B 24.942,C -1.7587,E1 24.9262,E2 692.7787} C_DIS
LIN {X -59.7019,Y 107.3297,Z 135,A 115.4296,B 24.9423,C -1.7546,E1 24.9211,E2 690.6954} C_DIS
LIN {X -63.3606,Y 105.2112,Z 135,A 117.3965,B 24.9426,C -1.7507,E1 24.9164,E2 688.7318} C_DIS
LIN {X -67.0227,Y 102.917,Z 135,A 119.4163,B 24.9428,C -1.747,E1 24.9116,E2 686.7143} C_DIS
LIN {X -70.3892,Y 100.6447,Z 135,A 121.1893,B 24.9434,C -1.7377,E1 24.9076,E2 684.9575} C_DIS
LIN {X -74.1526,Y 97.9048,Z 135,A 123.5223,B 24.9432,C -1.7404,E1 24.9023,E2 682.6098} C_DIS
LIN {X -77.5033,Y 95.2745,Z 135,A 125.5367,B 24.9434,C -1.7372,E1 24.8979,E2 680.5955} C_DIS
LIN {X -80.9745,Y 92.3425,Z 135,A 127.3511,B 24.9446,C -1.7188,E1 24.8942,E2 678.818} C_DIS
LIN {X -83.591,Y 89.9804,Z 135,A 129.2637,B 24.9441,C -1.7268,E1 24.8902,E2 676.8785} C_DIS
LIN {X -86.529,Y 87.1588,Z 135,A 131.2106,B 24.9443,C -1.7243,E1 24.8863,E2 674.9294} C_DIS
LIN {X -89.6295,Y 83.9678,Z 135,A 133.3284,B 24.9445,C -1.7209,E1 24.8822,E2 672.8105} C_DIS
LIN {X -92.6262,Y 80.6493,Z 135,A 135.3856,B 24.9449,C -1.7143,E1 24.8784,E2 670.7598} C_DIS
LIN {X -95.2794,Y 77.4973,Z 135,A 137.3209,B 24.9452,C -1.7098,E1 24.8749,E2 668.8264} C_DIS
LIN {X -97.8281,Y 74.2542,Z 135,A 139.288,B 24.9454,C -1.7064,E1 24.8716,E2 666.8579} C_DIS
LIN {X -100.2225,Y 70.9889,Z 135,A 141.1726,B 24.9458,C -1.701,E1 24.8685,E2 664.977} C_DIS
LIN {X -102.7477,Y 67.2824,Z 135,A 143.0707,B 24.9467,C -1.6865,E1 24.8656,E2 663.104} C_DIS
LIN {X -104.6063,Y 64.3542,Z 135,A 144.8741,B 24.9465,C -1.69,E1 24.8629,E2 661.2831} C_DIS
LIN {X -107.5135,Y 59.3693,Z 135,A 147.8269,B 24.9462,C -1.6936,E1 24.8588,E2 658.3063} C_DIS
LIN {X -110.6781,Y 53.2347,Z 135,A 150.7748,B 24.9476,C -1.6719,E1 24.8552,E2 655.3944} C_DIS
LIN {X -111.8893,Y 50.6414,Z 135,A 152.2076,B 24.9476,C -1.672,E1 24.8535,E2 653.9532} C_DIS
LIN {X -113.2946,Y 47.4112,Z 135,A 153.7403,B 24.9482,C -1.6621,E1 24.8518,E2 652.4358} C_DIS
LIN {X -114.4613,Y 44.5207,Z 135,A 155.1522,B 24.9486,C -1.6557,E1 24.8504,E2 651.0312} C_DIS
LIN {X -115.5338,Y 41.6583,Z 135,A 156.6298,B 24.9488,C -1.6535,E1 24.849,E2 649.5505} C_DIS
LIN {X -116.6215,Y 38.5099,Z 135,A 158.2152,B 24.949,C -1.6499,E1 24.8475,E2 647.9646} C_DIS
LIN {X -117.8242,Y 34.6551,Z 135,A 160.1152,B 24.9493,C -1.6446,E1 24.846,E2 646.0663} C_DIS
LIN {X -118.7259,Y 31.4281,Z 135,A 161.6968,B 24.9496,C -1.6404,E1 24.8448,E2 644.4855} C_DIS
LIN {X -119.8199,Y 26.9605,Z 135,A 163.8113,B 24.9501,C -1.6321,E1 24.8435,E2 642.3784} C_DIS
LIN {X -120.8615,Y 21.8189,Z 135,A 166.3196,B 24.9504,C -1.6268,E1 24.8421,E2 639.868} C_DIS
LIN {X -121.416,Y 18.4875,Z 135,A 167.9782,B 24.9505,C -1.6253,E1 24.8414,E2 638.2032} C_DIS
LIN {X -121.8654,Y 15.259,Z 135,A 169.6468,B 24.9505,C -1.6268,E1 24.8408,E2 636.521} C_DIS
LIN {X -122.5916,Y 7.4092,Z 135,A 172.715,B 24.9528,C -1.588,E1 24.8401,E2 633.5268} C_DIS
LIN {X -122.7538,Y 3.9112,Z 135,A 174.9571,B 24.9515,C -1.6092,E1 24.8398,E2 631.2206} C_DIS
LIN {X -122.7495,Y -4.0725,Z 135,A 178.4605,B 24.9528,C -1.5872,E1 24.8399,E2 627.7486} C_DIS
LIN {X -122.4568,Y -9.3804,Z 135,A -178.8224,B 24.9527,C -1.5896,E1 24.8404,E2 625.0096} C_DIS
LIN {X -121.6697,Y -16.7458,Z 135,A -175.4153,B 24.9534,C -1.5762,E1 24.8415,E2 621.6139} C_DIS
LIN {X -121.0237,Y -20.9119,Z 135,A -172.6503,B 24.9517,C -1.6054,E1 24.8429,E2 618.7629} C_DIS
LIN {X -119.9096,Y -26.5641,Z 135,A -170.7001,B 24.9542,C -1.5641,E1 24.8439,E2 616.8998} C_DIS
LIN {X -119.0652,Y -30.1164,Z 135,A -169.0356,B 24.9546,C -1.557,E1 24.845,E2 615.2423} C_DIS
LIN {X -117.9802,Y -34.1224,Z 135,A -167.1057,B 24.9549,C -1.5508,E1 24.8465,E2 613.3161} C_DIS
LIN {X -116.9611,Y -37.4647,Z 135,A -165.4549,B 24.9552,C -1.5467,E1 24.8479,E2 611.6656} C_DIS
LIN {X -113.8177,Y -46.1418,Z 135,A -161.1781,B 24.956,C -1.5324,E1 24.852,E2 607.3987} C_DIS
LIN {X -110.6997,Y -53.1894,Z 135,A -157.4861,B 24.9564,C -1.5262,E1 24.8563,E2 603.7011} C_DIS
LIN {X -108.8496,Y -56.8794,Z 135,A -155.6275,B 24.9568,C -1.5178,E1 24.8586,E2 601.8527} C_DIS
LIN {X -107.4625,Y -59.462,Z 135,A -153.5768,B 24.9553,C -1.5446,E1 24.8615,E2 599.7272} C_DIS
LIN {X -105.0486,Y -63.6294,Z 135,A -152.1826,B 24.9578,C -1.5003,E1 24.8634,E2 598.4315} C_DIS
LIN {X -101.9305,Y -68.5145,Z 135,A -149.1419,B 24.9574,C -1.5082,E1 24.868,E2 595.3566} C_DIS
LIN {X -99.5408,Y -71.9414,Z 135,A -147.2523,B 24.9578,C -1.5006,E1 24.871,E2 593.4759} C_DIS
LIN {X -97.4075,Y -74.8047,Z 135,A -145.5953,B 24.9581,C -1.496,E1 24.8738,E2 591.8218} C_DIS
LIN {X -95.204,Y -77.5893,Z 135,A -143.8628,B 24.9581,C -1.4955,E1 24.8769,E2 590.0826} C_DIS
LIN {X -92.3212,Y -80.9988,Z 135,A -141.8332,B 24.9585,C -1.4882,E1 24.8806,E2 588.0611} C_DIS
LIN {X -89.5974,Y -84.0022,Z 135,A -139.8884,B 24.9586,C -1.4863,E1 24.8842,E2 586.1122} C_DIS
LIN {X -87.1891,Y -86.4984,Z 135,A -138.2258,B 24.9586,C -1.4848,E1 24.8875,E2 584.446} C_DIS
LIN {X -84.0128,Y -89.5874,Z 135,A -136.1325,B 24.9589,C -1.4817,E1 24.8917,E2 582.3516} C_DIS
LIN {X -80.883,Y -92.4223,Z 135,A -134.1979,B 24.9592,C -1.4761,E1 24.8958,E2 580.4225} C_DIS
LIN {X -77.8036,Y -95.0291,Z 135,A -132.4119,B 24.9596,C -1.4681,E1 24.8996,E2 578.6488} C_DIS
LIN {X -75.0114,Y -97.2485,Z 135,A -130.6493,B 24.9596,C -1.4695,E1 24.9035,E2 576.8762} C_DIS
LIN {X -72.7206,Y -98.9728,Z 135,A -128.9117,B 24.9587,C -1.4856,E1 24.9075,E2 575.0943} C_DIS
LIN {X -69.5328,Y -101.2378,Z 135,A -127.5076,B 24.9599,C -1.4631,E1 24.9106,E2 573.7388} C_DIS
LIN {X -67.0023,Y -102.9302,Z 135,A -125.5519,B 24.9587,C -1.4856,E1 24.9153,E2 571.7233} C_DIS
LIN {X -63.2487,Y -105.2789,Z 135,A -123.9671,B 24.9601,C -1.4602,E1 24.919,E2 570.1941} C_DIS
LIN {X -59.7514,Y -107.3022,Z 135,A -122.0505,B 24.9601,C -1.459,E1 24.9236,E2 568.2747} C_DIS
LIN {X -56.6639,Y -108.9628,Z 135,A -120.5254,B 24.9605,C -1.4517,E1 24.9274,E2 566.7627} C_DIS
LIN {X -53.0957,Y -110.7445,Z 135,A -118.6948,B 24.9607,C -1.448,E1 24.9319,E2 564.9361} C_DIS
LIN {X -49.2987,Y -112.4867,Z 135,A -116.3653,B 24.9599,C -1.4636,E1 24.938,E2 562.5641} C_DIS
LIN {X -46.2761,Y -113.7636,Z 135,A -115.1387,B 24.9607,C -1.4477,E1 24.9411,E2 561.3722} C_DIS
LIN {X -43.0909,Y -115.0072,Z 135,A -113.6117,B 24.961,C -1.443,E1 24.945,E2 559.8532} C_DIS
LIN {X -40.1272,Y -116.0746,Z 135,A -111.7948,B 24.9602,C -1.4581,E1 24.9499,E2 557.9971} C_DIS
LIN {X -35.4029,Y -117.6029,Z 135,A -109.6874,B 24.9608,C -1.4464,E1 24.9555,E2 555.9136} C_DIS
LIN {X -31.9693,Y -118.5815,Z 135,A -108.2379,B 24.9614,C -1.4352,E1 24.9593,E2 554.4885} C_DIS
LIN {X -28.8319,Y -119.3828,Z 135,A -106.5687,B 24.9611,C -1.4418,E1 24.9639,E2 552.8013} C_DIS
LIN {X -24.8148,Y -120.2824,Z 135,A -104.8458,B 24.9616,C -1.4316,E1 24.9685,E2 551.1006} C_DIS
LIN {X -19.0034,Y -121.3361,Z 135,A -102.0452,B 24.9616,C -1.4327,E1 24.9763,E2 548.2944} C_DIS
LIN {X -16.0524,Y -121.7616,Z 135,A -100.534,B 24.9613,C -1.4381,E1 24.9805,E2 546.7692} C_DIS
LIN {X -12.3278,Y -122.1963,Z 135,A -98.7075,B 24.9611,C -1.4415,E1 24.9856,E2 544.9335} C_DIS
LIN {X -8.7575,Y -122.5027,Z 135,A -97.0037,B 24.961,C -1.4431,E1 24.9903,E2 543.2253} C_DIS
LIN {X -4.8344,Y -122.7201,Z 135,A -95.2535,B 24.9612,C -1.4392,E1 24.9952,E2 541.4837} C_DIS
LIN {X -0.8318,Y -122.8126,Z 135,A -93.4409,B 24.9613,C -1.4369,E1 25.0002,E2 539.6766} C_DIS
LIN {X -0.8318,Y -122.8126,Z 135,A -93.4409,B 24.9613,C -1.4369,E1 25.0002,E2 539.6766} C_DIS
Enddeposition()
LIN {X 0.8577,Y -121.8167,Z 135,A -92.8543,B 24.9609,C -1.4448,E1 25.0019,E2 539.0713} C_DIS
Startdeposition()
$VEL.CP = VEL_PRINT
LIN {X -1.9004,Y -121.8077,Z 135,A -94.706,B 24.9623,C -1.4183,E1 24.9966,E2 540.9857} C_DIS
LIN {X -6.0387,Y -121.6727,Z 135,A -96.5811,B 24.9621,C -1.4215,E1 24.9913,E2 542.8537} C_DIS
LIN {X -9.8764,Y -121.422,Z 135,A -98.4461,B 24.9623,C -1.4189,E1 24.9861,E2 544.7256} C_DIS
LIN {X -13.3169,Y -121.0926,Z 135,A -100.1495,B 24.9625,C -1.4155,E1 24.9814,E2 546.4381} C_DIS
LIN {X -17.8995,Y -120.502,Z 135,A -102.7302,B 24.9634,C -1.3971,E1 24.9741,E2 549.0644} C_DIS
LIN {X -21.9265,Y -119.8337,Z 135,A -104.1498,B 24.9622,C -1.4208,E1 24.9704,E2 550.4292} C_DIS
LIN {X -26.768,Y -118.8455,Z 135,A -106.2564,B 24.9616,C -1.4319,E1 24.9647,E2 552.5119} C_DIS
LIN {X -29.7894,Y -118.1239,Z 135,A -107.9953,B 24.9622,C -1.4199,E1 24.9599,E2 554.2818} C_DIS
LIN {X -32.8948,Y -117.2969,Z 135,A -109.4268,B 24.962,C -1.4246,E1 24.956,E2 555.7045} C_DIS
LIN {X -36.3461,Y -116.276,Z 135,A -111.085,B 24.9618,C -1.4273,E1 24.9516,E2 557.3589} C_DIS
LIN {X -39.5243,Y -115.2329,Z 135,A -112.7899,B 24.9621,C -1.4226,E1 24.9471,E2 559.0782} C_DIS
LIN {X -42.9855,Y -113.9865,Z 135,A -114.5059,B 24.962,C -1.4249,E1 24.9426,E2 560.7924} C_DIS
LIN {X -49.6252,Y -111.2563,Z 135,A -117.519,B 24.9609,C -1.445,E1 24.9349,E2 563.7645} C_DIS
LIN {X -51.8568,Y -110.2361,Z 135,A -119.3508,B 24.9625,C -1.4156,E1 24.9301,E2 565.6708} C_DIS
LIN {X -54.8534,Y -108.7745,Z 135,A -120.3921,B 24.9611,C -1.4414,E1 24.9276,E2 566.6536} C_DIS
LIN {X -57.6805,Y -107.3033,Z 135,A -122.019,B 24.9613,C -1.4375,E1 24.9236,E2 568.2941} C_DIS
LIN {X -60.7134,Y -105.6175,Z 135,A -123.8162,B 24.9616,C -1.4324,E1 24.9192,E2 570.1088} C_DIS
LIN {X -65.5671,Y -102.6743,Z 135,A -126.2665,B 24.9608,C -1.4463,E1 24.9134,E2 572.5337} C_DIS
LIN {X -68.436,Y -100.7848,Z 135,A -128.3551,B 24.9618,C -1.4278,E1 24.9084,E2 574.6732} C_DIS
LIN {X -71.2313,Y -98.8294,Z 135,A -129.7229,B 24.9611,C -1.4411,E1 24.9054,E2 576.0142} C_DIS
LIN {X -74.8627,Y -96.1078,Z 135,A -132.0036,B 24.9612,C -1.4384,E1 24.9003,E2 578.3094} C_DIS
LIN {X -78.4839,Y -93.1739,Z 135,A -134.0389,B 24.9606,C -1.4496,E1 24.896,E2 580.3259} C_DIS
LIN {X -81.6417,Y -90.4199,Z 135,A -136.0344,B 24.9605,C -1.4524,E1 24.8918,E2 582.3226} C_DIS
LIN {X -84.8066,Y -87.4579,Z 135,A -138.0546,B 24.9602,C -1.4575,E1 24.8877,E2 584.339} C_DIS
LIN {X -87.7828,Y -84.471,Z 135,A -140.0793,B 24.9601,C -1.46,E1 24.8838,E2 586.3664} C_DIS
LIN {X -90.9465,Y -81.0546,Z 135,A -142.253,B 24.9598,C -1.4657,E1 24.8797,E2 588.5363} C_DIS
LIN {X -93.6706,Y -77.8904,Z 135,A -144.4867,B 24.9601,C -1.4585,E1 24.8756,E2 590.7973} C_DIS
LIN {X -95.7426,Y -75.3286,Z 135,A -145.4755,B 24.9586,C -1.4869,E1 24.874,E2 591.7233} C_DIS
LIN {X -97.4832,Y -73.063,Z 135,A -147.1587,B 24.9592,C -1.4753,E1 24.8711,E2 593.4421} C_DIS
LIN {X -99.9267,Y -69.6828,Z 135,A -149.1091,B 24.9589,C -1.4808,E1 24.8679,E2 595.3889} C_DIS
LIN {X -102.529,Y -65.794,Z 135,A -151.2079,B 24.9584,C -1.491,E1 24.8647,E2 597.474} C_DIS
LIN {X -104.2153,Y -63.0889,Z 135,A -152.7239,B 24.9582,C -1.4943,E1 24.8625,E2 598.9899} C_DIS
LIN {X -106.3615,Y -59.4001,Z 135,A -154.8212,B 24.9581,C -1.4958,E1 24.8596,E2 601.0945} C_DIS
LIN {X -108.0515,Y -56.2638,Z 135,A -156.4243,B 24.9576,C -1.5037,E1 24.8575,E2 602.6874} C_DIS
LIN {X -109.7625,Y -52.8481,Z 135,A -158.6648,B 24.9584,C -1.4896,E1 24.8547,E2 604.9735} C_DIS
LIN {X -111.2658,Y -49.6038,Z 135,A -159.9268,B 24.9571,C -1.5126,E1 24.8533,E2 606.1876} C_DIS
LIN {X -112.5679,Y -46.575,Z 135,A -161.4863,B 24.9569,C -1.5167,E1 24.8516,E2 607.7459} C_DIS
LIN {X -113.9861,Y -42.9867,Z 135,A -163.7698,B 24.9577,C -1.502,E1 24.8493,E2 610.0775} C_DIS
LIN {X -115.2639,Y -39.4347,Z 135,A -165.0548,B 24.9562,C -1.5284,E1 24.8482,E2 611.3068} C_DIS
LIN {X -116.0558,Y -37.0361,Z 135,A -166.3018,B 24.9562,C -1.5295,E1 24.8471,E2 612.5584} C_DIS
LIN {X -117.1373,Y -33.4657,Z 135,A -168.2444,B 24.9563,C -1.5268,E1 24.8456,E2 614.5187} C_DIS
LIN {X -118.1369,Y -29.7383,Z 135,A -169.8705,B 24.9555,C -1.5406,E1 24.8444,E2 616.1213} C_DIS
LIN {X -118.9912,Y -26.1137,Z 135,A -172.0204,B 24.9562,C -1.529,E1 24.8431,E2 618.3114} C_DIS
LIN {X -119.6467,Y -22.9201,Z 135,A -173.1259,B 24.9549,C -1.5522,E1 24.8425,E2 619.3682} C_DIS
LIN {X -120.1863,Y -19.8983,Z 135,A -174.7282,B 24.9549,C -1.55,E1 24.8418,E2 620.9852} C_DIS
LIN {X -120.7817,Y -15.8888,Z 135,A -176.7963,B 24.955,C -1.5492,E1 24.8409,E2 623.0675} C_DIS
LIN {X -121.3241,Y -11.0248,Z 135,A -179.5793,B 24.9558,C -1.5362,E1 24.8403,E2 625.8983} C_DIS
LIN {X -121.6604,Y -6.2833,Z 135,A 178.8905,B 24.9536,C -1.5735,E1 24.84,E2 627.3488} C_DIS
LIN {X -121.7907,Y -2.8371,Z 135,A 176.5153,B 24.9552,C -1.5467,E1 24.8398,E2 629.802} C_DIS
LIN {X -121.8057,Y 2.0227,Z 135,A 174.5928,B 24.9538,C -1.5696,E1 24.8398,E2 631.6817} C_DIS
LIN {X -121.7107,Y 5.2394,Z 135,A 173.4538,B 24.9526,C -1.5905,E1 24.84,E2 632.7777} C_DIS
LIN {X -121.5175,Y 8.6176,Z 135,A 171.5152,B 24.9532,C -1.5809,E1 24.8403,E2 634.7507} C_DIS
LIN {X -121.1404,Y 12.8735,Z 135,A 169.7306,B 24.9522,C -1.5971,E1 24.8408,E2 636.5075} C_DIS
LIN {X -120.7623,Y 16.0374,Z 135,A 168.2484,B 24.9519,C -1.6027,E1 24.8413,E2 637.9852} C_DIS
LIN {X -120.2856,Y 19.2999,Z 135,A 166.5967,B 24.9519,C -1.6034,E1 24.842,E2 639.645} C_DIS
LIN {X -119.6343,Y 22.9851,Z 135,A 164.8845,B 24.9514,C -1.6112,E1 24.8429,E2 641.3488} C_DIS
LIN {X -118.9177,Y 26.4519,Z 135,A 163.05,B 24.9514,C -1.6094,E1 24.844,E2 643.1984} C_DIS
LIN {X -117.9108,Y 30.6293,Z 135,A 161.0729,B 24.951,C -1.6178,E1 24.8453,E2 645.1671} C_DIS
LIN {X -116.917,Y 34.2206,Z 135,A 159.4275,B 24.9503,C -1.628,E1 24.8466,E2 646.7977} C_DIS
LIN {X -115.7871,Y 37.8733,Z 135,A 157.5175,B 24.9503,C -1.6289,E1 24.8482,E2 648.7164} C_DIS
LIN {X -114.601,Y 41.3185,Z 135,A 155.9418,B 24.9496,C -1.6402,E1 24.8496,E2 650.274} C_DIS
LIN {X -113.5279,Y 44.1818,Z 135,A 154.4703,B 24.9494,C -1.6433,E1 24.8511,E2 651.7465} C_DIS
LIN {X -112.0625,Y 47.7805,Z 135,A 152.5033,B 24.9494,C -1.643,E1 24.8532,E2 653.7252} C_DIS
LIN {X -110.5026,Y 51.2816,Z 135,A 150.766,B 24.9489,C -1.6513,E1 24.8552,E2 655.4522} C_DIS
LIN {X -108.7991,Y 54.8053,Z 135,A 148.5128,B 24.9496,C -1.6393,E1 24.8581,E2 657.7462} C_DIS
LIN {X -107.0563,Y 58.1381,Z 135,A 146.6575,B 24.9496,C -1.6408,E1 24.8606,E2 659.6075} C_DIS
LIN {X -105.0687,Y 61.6573,Z 135,A 145.4063,B 24.9475,C -1.6742,E1 24.8622,E2 660.7857} C_DIS
LIN {X -102.5242,Y 65.8016,Z 135,A 142.986,B 24.9475,C -1.6751,E1 24.8658,E2 663.2164} C_DIS
LIN {X -100.8654,Y 68.3169,Z 135,A 141.4526,B 24.9475,C -1.6741,E1 24.8682,E2 664.7598} C_DIS
LIN {X -98.4199,Y 71.7962,Z 135,A 139.3772,B 24.9473,C -1.6764,E1 24.8716,E2 666.8399} C_DIS
LIN {X -95.7693,Y 75.2946,Z 135,A 137.3529,B 24.9469,C -1.6837,E1 24.875,E2 668.8562} C_DIS
LIN {X -93.1197,Y 78.5485,Z 135,A 135.364,B 24.9466,C -1.6883,E1 24.8785,E2 670.8435} C_DIS
LIN {X -90.4609,Y 81.5965,Z 135,A 133.4116,B 24.9464,C -1.691,E1 24.8822,E2 672.7981} C_DIS
LIN {X -87.3809,Y 84.8862,Z 135,A 131.3393,B 24.9459,C -1.6984,E1 24.8861,E2 674.8619} C_DIS
LIN {X -84.7212,Y 87.5406,Z 135,A 129.553,B 24.9457,C -1.7019,E1 24.8897,E2 676.6474} C_DIS
LIN {X -81.6381,Y 90.4232,Z 135,A 127.5549,B 24.9455,C -1.706,E1 24.8938,E2 678.6438} C_DIS
LIN {X -78.5903,Y 93.0846,Z 135,A 125.5902,B 24.9454,C -1.7076,E1 24.898,E2 680.6121} C_DIS
LIN {X -75.2701,Y 95.7886,Z 135,A 123.6136,B 24.945,C -1.7137,E1 24.9023,E2 682.5817} C_DIS
LIN {X -71.7444,Y 98.4575,Z 135,A 121.6945,B 24.9442,C -1.7251,E1 24.9065,E2 684.4805} C_DIS
LIN {X -69.1379,Y 100.3047,Z 135,A 119.9818,B 24.9446,C -1.719,E1 24.9105,E2 686.2137} C_DIS
LIN {X -65.4587,Y 102.7437,Z 135,A 117.9321,B 24.9443,C -1.7242,E1 24.9153,E2 688.2577} C_DIS
LIN {X -62.0537,Y 104.8356,Z 135,A 115.9968,B 24.9443,C -1.7252,E1 24.9199,E2 690.1964} C_DIS
LIN {X -58.133,Y 107.0591,Z 135,A 113.6441,B 24.9446,C -1.7187,E1 24.9257,E2 692.5713} C_DIS
LIN {X -54.5867,Y 108.9103,Z 135,A 111.9995,B 24.9438,C -1.7322,E1 24.9297,E2 694.1882} C_DIS
LIN {X -51.1334,Y 110.5711,Z 135,A 110.3121,B 24.9432,C -1.7402,E1 24.934,E2 695.8609} C_DIS
LIN {X -47.636,Y 112.1248,Z 135,A 108.5377,B 24.943,C -1.744,E1 24.9385,E2 697.6306} C_DIS
LIN {X -43.2374,Y 113.8922,Z 135,A 106.1525,B 24.9432,C -1.7401,E1 24.9447,E2 700.0301} C_DIS
LIN {X -39.5928,Y 115.2091,Z 135,A 104.4241,B 24.9428,C -1.7467,E1 24.9492,E2 701.7464} C_DIS
LIN {X -34.926,Y 116.7103,Z 135,A 102.1781,B 24.9425,C -1.752,E1 24.9552,E2 703.9836} C_DIS
LIN {X -32.0851,Y 117.5231,Z 135,A 100.6064,B 24.9429,C -1.7453,E1 24.9595,E2 705.5737} C_DIS
LIN {X -28.3343,Y 118.4815,Z 135,A 98.6303,B 24.9432,C -1.7402,E1 24.9649,E2 707.5648} C_DIS
LIN {X -24.8438,Y 119.2634,Z 135,A 97.1891,B 24.9424,C -1.7524,E1 24.9687,E2 708.9786} C_DIS
LIN {X -18.7765,Y 120.3667,Z 135,A 94.352,B 24.9421,C -1.7575,E1 24.9765,E2 711.8065} C_DIS
LIN {X -15.7296,Y 120.8026,Z 135,A 92.8534,B 24.9422,C -1.7561,E1 24.9807,E2 713.3096} C_DIS
LIN {X -11.5535,Y 121.2733,Z 135,A 90.8911,B 24.9421,C -1.7578,E1 24.9861,E2 715.269} C_DIS
LIN {X -4.3978,Y 121.7436,Z 135,A 87.4729,B 24.9421,C -1.757,E1 24.9957,E2 718.6901} C_DIS
LIN {X 0.0146,Y 121.8243,Z 135,A 85.3162,B 24.9424,C -1.7538,E1 25.0017,E2 720.8546} C_DIS
LIN {X 3.7515,Y 121.7653,Z 135,A 83.5637,B 24.9424,C -1.7542,E1 25.0066,E2 722.6056} C_DIS
LIN {X 8.1161,Y 121.5534,Z 135,A 81.504,B 24.9424,C -1.754,E1 25.0123,E2 724.665} C_DIS
LIN {X 13.892,Y 121.0289,Z 135,A 79.0182,B 24.9416,C -1.7649,E1 25.0192,E2 727.1236} C_DIS
LIN {X 18.1267,Y 120.4673,Z 135,A 77.0196,B 24.9416,C -1.7649,E1 25.0247,E2 729.1205} C_DIS
LIN {X 23.6105,Y 119.5141,Z 135,A 74.3401,B 24.9419,C -1.761,E1 25.0321,E2 731.8064} C_DIS
LIN {X 25.762,Y 119.0671,Z 135,A 73.1883,B 24.9423,C -1.755,E1 25.0352,E2 732.9708} C_DIS
LIN {X 28.8891,Y 118.3477,Z 135,A 71.7799,B 24.942,C -1.7588,E1 25.039,E2 734.3681} C_DIS
LIN {X 32.0857,Y 117.523,Z 135,A 70.2229,B 24.9421,C -1.7576,E1 25.0432,E2 735.9256} C_DIS
LIN {X 34.8274,Y 116.7393,Z 135,A 68.647,B 24.9429,C -1.7456,E1 25.0475,E2 737.5272} C_DIS
LIN {X 38.5461,Y 115.5631,Z 135,A 67.0223,B 24.9423,C -1.754,E1 25.0518,E2 739.129} C_DIS
LIN {X 41.9241,Y 114.3827,Z 135,A 64.2762,B 24.9457,C -1.7028,E1 25.0593,E2 741.9905} C_DIS
LIN {X 48.0534,Y 111.9445,Z 135,A 62.4524,B 24.942,C -1.7593,E1 25.0637,E2 743.6763} C_DIS
LIN {X 52.6093,Y 109.8766,Z 135,A 59.8763,B 24.9429,C -1.7459,E1 25.0703,E2 746.2776} C_DIS
LIN {X 56.2183,Y 108.0754,Z 135,A 57.9773,B 24.943,C -1.7433,E1 25.075,E2 748.1776} C_DIS
LIN {X 59.6769,Y 106.206,Z 135,A 55.2546,B 24.9459,C -1.6994,E1 25.0819,E2 750.996} C_DIS
LIN {X 64.7705,Y 103.179,Z 135,A 52.9911,B 24.9446,C -1.7197,E1 25.0871,E2 753.2043} C_DIS
LIN {X 67.6692,Y 101.3011,Z 135,A 51.8849,B 24.9431,C -1.7418,E1 25.0895,E2 754.2546} C_DIS
LIN {X 70.0511,Y 99.6691,Z 135,A 50.3103,B 24.944,C -1.7291,E1 25.0932,E2 755.8539} C_DIS
LIN {X 73.6356,Y 97.0512,Z 135,A 48.2244,B 24.9442,C -1.7254,E1 25.0979,E2 757.941} C_DIS
LIN {X 76.9343,Y 94.4573,Z 135,A 46.4527,B 24.9438,C -1.7315,E1 25.1017,E2 759.6918} C_DIS
LIN {X 79.5391,Y 92.2744,Z 135,A 44.6986,B 24.9445,C -1.7208,E1 25.1055,E2 761.4643} C_DIS
LIN {X 82.4704,Y 89.6642,Z 135,A 42.6798,B 24.9453,C -1.7087,E1 25.1097,E2 763.5036} C_DIS
LIN {X 86.1729,Y 86.1127,Z 135,A 40.3959,B 24.9453,C -1.7097,E1 25.1142,E2 765.7755} C_DIS
LIN {X 89.3254,Y 82.8376,Z 135,A 38.3054,B 24.9453,C -1.7072,E1 25.1182,E2 767.8628} C_DIS
LIN {X 92.1108,Y 79.7291,Z 135,A 36.3791,B 24.9456,C -1.7044,E1 25.1218,E2 769.787} C_DIS
LIN {X 94.8554,Y 76.4427,Z 135,A 34.3735,B 24.9458,C -1.7,E1 25.1253,E2 771.7938} C_DIS
LIN {X 97.326,Y 73.2715,Z 135,A 32.5053,B 24.9461,C -1.6964,E1 25.1285,E2 773.6616} C_DIS
LIN {X 101.2596,Y 67.7315,Z 135,A 29.4291,B 24.9462,C -1.694,E1 25.1334,E2 776.7284} C_DIS
LIN {X 102.806,Y 65.3614,Z 135,A 27.9192,B 24.947,C -1.6817,E1 25.1357,E2 778.2597} C_DIS
LIN {X 105.2009,Y 61.4322,Z 135,A 25.8219,B 24.9472,C -1.6792,E1 25.1387,E2 780.3524} C_DIS
LIN {X 107.1806,Y 57.9089,Z 135,A 23.975,B 24.9473,C -1.6765,E1 25.1412,E2 782.1958} C_DIS
LIN {X 108.5701,Y 55.255,Z 135,A 22.617,B 24.9474,C -1.6751,E1 25.1429,E2 783.5499} C_DIS
LIN {X 110.2991,Y 51.7216,Z 135,A 20.6413,B 24.9481,C -1.6636,E1 25.1453,E2 785.5422} C_DIS
LIN {X 111.7198,Y 48.573,Z 135,A 19.1556,B 24.9481,C -1.6657,E1 25.147,E2 787.0148} C_DIS
LIN {X 113.0554,Y 45.3775,Z 135,A 17.5358,B 24.9483,C -1.6614,E1 25.1487,E2 788.636} C_DIS
LIN {X 114.2526,Y 42.2751,Z 135,A 16.0532,B 24.9483,C -1.6607,E1 25.1502,E2 790.1118} C_DIS
LIN {X 115.3443,Y 39.2029,Z 135,A 14.3283,B 24.9492,C -1.6465,E1 25.1518,E2 791.8604} C_DIS
LIN {X 116.8319,Y 34.5112,Z 135,A 12.1249,B 24.9492,C -1.645,E1 25.1536,E2 794.0549} C_DIS
LIN {X 117.8243,Y 30.956,Z 135,A 10.4715,B 24.9494,C -1.6437,E1 25.1548,E2 795.7019} C_DIS
LIN {X 118.96,Y 26.2579,Z 135,A 7.4979,B 24.9519,C -1.6019,E1 25.1567,E2 798.7568} C_DIS
LIN {X 119.9112,Y 21.4936,Z 135,A 5.8468,B 24.9505,C -1.6259,E1 25.1575,E2 800.3415} C_DIS
LIN {X 120.4647,Y 18.1435,Z 135,A 3.8653,B 24.9519,C -1.6017,E1 25.1584,E2 802.3685} C_DIS
LIN {X 120.9706,Y 14.3808,Z 135,A 2.5334,B 24.9509,C -1.6185,E1 25.1588,E2 803.6529} C_DIS
LIN {X 121.3781,Y 10.3956,Z 135,A 0.6451,B 24.9513,C -1.6122,E1 25.1593,E2 805.545} C_DIS
LIN {X 121.6578,Y 6.3351,Z 135,A -1.2521,B 24.9516,C -1.6068,E1 25.1596,E2 807.4436} C_DIS
LIN {X 121.7999,Y 2.3743,Z 135,A -3.0964,B 24.9519,C -1.6016,E1 25.1598,E2 809.289} C_DIS
LIN {X 121.8181,Y -1.1883,Z 135,A -4.8456,B 24.9525,C -1.5924,E1 25.1598,E2 811.0495} C_DIS
LIN {X 121.724,Y -4.8987,Z 135,A -6.5001,B 24.9525,C -1.5913,E1 25.1596,E2 812.697} C_DIS
LIN {X 121.5009,Y -8.8446,Z 135,A -8.7065,B 24.9539,C -1.5679,E1 25.1592,E2 814.9454} C_DIS
LIN {X 121.1865,Y -12.4429,Z 135,A -10.7353,B 24.9552,C -1.5459,E1 25.1586,E2 817.0139} C_DIS
LIN {X 120.5566,Y -17.5175,Z 135,A -12.2258,B 24.953,C -1.5835,E1 25.1581,E2 818.4071} C_DIS
LIN {X 120.0102,Y -20.9363,Z 135,A -14.2352,B 24.9545,C -1.5591,E1 25.1571,E2 820.4621} C_DIS
LIN {X 119.2053,Y -25.122,Z 135,A -16.394,B 24.9553,C -1.5449,E1 25.1559,E2 822.6419} C_DIS
LIN {X 118.445,Y -28.4854,Z 135,A -17.3398,B 24.9536,C -1.5734,E1 25.1553,E2 823.5149} C_DIS
LIN {X 117.7936,Y -31.071,Z 135,A -18.8981,B 24.9547,C -1.5541,E1 25.1542,E2 825.1098} C_DIS
LIN {X 116.7568,Y -34.7677,Z 135,A -20.9582,B 24.9558,C -1.5356,E1 25.1526,E2 827.2017} C_DIS
LIN {X 115.8039,Y -37.823,Z 135,A -22.0862,B 24.955,C -1.5496,E1 25.1517,E2 828.2903} C_DIS
LIN {X 114.3605,Y -41.9857,Z 135,A -24.3222,B 24.9559,C -1.5348,E1 25.1495,E2 830.5486} C_DIS
LIN {X 111.4605,Y -49.1686,Z 135,A -27.7326,B 24.9559,C -1.5351,E1 25.146,E2 833.9395} C_DIS
LIN {X 109.807,Y -52.7549,Z 135,A -29.609,B 24.9562,C -1.5285,E1 25.1437,E2 835.8215} C_DIS
LIN {X 107.1905,Y -57.8905,Z 135,A -32.3968,B 24.9569,C -1.5164,E1 25.1401,E2 838.623} C_DIS
LIN {X 105.2918,Y -61.276,Z 135,A -34.1828,B 24.9571,C -1.5129,E1 25.1377,E2 840.4078} C_DIS
LIN {X 103.232,Y -64.6864,Z 135,A -36.1529,B 24.9577,C -1.5027,E1 25.1348,E2 842.3921} C_DIS
LIN {X 100.9466,Y -68.197,Z 135,A -37.956,B 24.9575,C -1.5054,E1 25.132,E2 844.18} C_DIS
LIN {X 98.93,Y -71.0914,Z 135,A -39.6793,B 24.958,C -1.4975,E1 25.1292,E2 845.9133} C_DIS
LIN {X 96.281,Y -74.6392,Z 135,A -41.8393,B 24.9585,C -1.4879,E1 25.1255,E2 848.0857} C_DIS
LIN {X 93.5948,Y -77.982,Z 135,A -43.8535,B 24.9588,C -1.4826,E1 25.122,E2 850.103} C_DIS
LIN {X 90.1707,Y -81.9163,Z 135,A -46.4892,B 24.9597,C -1.4673,E1 25.117,E2 852.7633} C_DIS
LIN {X 87.9559,Y -84.2901,Z 135,A -47.6024,B 24.9588,C -1.4838,E1 25.115,E2 853.8326} C_DIS
LIN {X 85.5562,Y -86.7255,Z 135,A -49.41,B 24.9595,C -1.4699,E1 25.1114,E2 855.6653} C_DIS
LIN {X 81.5065,Y -90.5413,Z 135,A -52.068,B 24.96,C -1.4617,E1 25.1059,E2 858.332} C_DIS
LIN {X 79.1135,Y -92.6399,Z 135,A -53.4634,B 24.9599,C -1.4632,E1 25.103,E2 859.7183} C_DIS
LIN {X 76.0655,Y -95.1585,Z 135,A -55.333,B 24.9602,C -1.4585,E1 25.0989,E2 861.5919} C_DIS
LIN {X 72.1612,Y -98.152,Z 135,A -57.4642,B 24.9599,C -1.4624,E1 25.0942,E2 863.7061} C_DIS
LIN {X 70.1596,Y -99.5926,Z 135,A -58.6157,B 24.96,C -1.4604,E1 25.0916,E2 864.8583} C_DIS
LIN {X 67.2062,Y -101.6092,Z 135,A -60.4123,B 24.9605,C -1.4514,E1 25.0874,E2 866.6702} C_DIS
LIN {X 64.3986,Y -103.4111,Z 135,A -61.9589,B 24.9606,C -1.4494,E1 25.0837,E2 868.2165} C_DIS
LIN {X 60.5021,Y -105.7382,Z 135,A -63.9423,B 24.9605,C -1.4528,E1 25.079,E2 870.1858} C_DIS
LIN {X 57.6182,Y -107.3368,Z 135,A -65.613,B 24.9609,C -1.4442,E1 25.0748,E2 871.8719} C_DIS
LIN {X 52.8285,Y -109.7719,Z 135,A -68.7173,B 24.9626,C -1.4122,E1 25.0669,E2 875.0436} C_DIS
LIN {X 48.6753,Y -111.6756,Z 135,A -70.0471,B 24.9607,C -1.4484,E1 25.0638,E2 876.2847} C_DIS
LIN {X 46.2754,Y -112.693,Z 135,A -71.7002,B 24.9619,C -1.4259,E1 25.0593,E2 877.9871} C_DIS
LIN {X 42.7942,Y -114.0582,Z 135,A -73.1836,B 24.9613,C -1.4367,E1 25.0556,E2 879.4416} C_DIS
LIN {X 39.484,Y -115.2468,Z 135,A -74.8764,B 24.9615,C -1.4327,E1 25.0511,E2 881.1405} C_DIS
LIN {X 35.8663,Y -116.4229,Z 135,A -76.8279,B 24.9621,C -1.4228,E1 25.0458,E2 883.112} C_DIS
LIN {X 30.9839,Y -117.8169,Z 135,A -78.9683,B 24.9616,C -1.432,E1 25.0401,E2 885.2271} C_DIS
LIN {X 28.0521,Y -118.5495,Z 135,A -80.5827,B 24.9622,C -1.4213,E1 25.0357,E2 886.8644} C_DIS
LIN {X 20.6238,Y -120.0652,Z 135,A -83.9115,B 24.9617,C -1.4295,E1 25.0267,E2 890.1698} C_DIS
LIN {X 13.3659,Y -121.0874,Z 135,A -87.2489,B 24.9616,C -1.4323,E1 25.0175,E2 893.4976} C_DIS
LIN {X 8.9349,Y -121.4943,Z 135,A -89.4905,B 24.962,C -1.4242,E1 25.0112,E2 895.7573} C_DIS
LIN {X 5.7488,Y -121.6873,Z 135,A -91.0065,B 24.962,C -1.4229,E1 25.0069,E2 897.2758} C_DIS
LIN {X 2.1053,Y -121.8043,Z 135,A -92.793,B 24.9623,C -1.419,E1 25.0019,E2 899.0713} C_DIS
LIN {X 2.1053,Y -121.8043,Z 135,A -92.793,B 24.9623,C -1.419,E1 25.0019,E2 899.0713} C_DIS
Enddeposition()
LIN {X 0.8485,Y -120.8246,Z 135,A -92.9224,B 24.9602,C -1.458,E1 25.0019,E2 899.1083} C_DIS
Startdeposition()
$VEL.CP = VEL_PRINT
LIN {X 4.0351,Y -120.7642,Z 135,A -91.073,B 24.9593,C -1.4743,E1 25.0071,E2 897.2204} C_DIS
LIN {X 7.8118,Y -120.5775,Z 135,A -89.432,B 24.9596,C -1.4679,E1 25.0116,E2 895.5953} C_DIS
LIN {X 10.8301,Y -120.3451,Z 135,A -87.8093,B 24.9591,C -1.4775,E1 25.0162,E2 893.9507} C_DIS
LIN {X 14.7579,Y -119.9258,Z 135,A -86.1267,B 24.9595,C -1.4696,E1 25.0208,E2 892.2881} C_DIS
LIN {X 17.9753,Y -119.4861,Z 135,A -84.6651,B 24.9597,C -1.4669,E1 25.0248,E2 890.8342} C_DIS
LIN {X 20.6479,Y -119.054,Z 135,A -83.2883,B 24.9594,C -1.4723,E1 25.0286,E2 889.4459} C_DIS
LIN {X 23.5386,Y -118.5159,Z 135,A -81.775,B 24.959,C -1.4792,E1 25.0328,E2 887.918} C_DIS
LIN {X 26.9083,Y -117.7951,Z 135,A -80.1905,B 24.959,C -1.4784,E1 25.0371,E2 886.3377} C_DIS
LIN {X 30.7776,Y -116.8444,Z 135,A -78.3857,B 24.9592,C -1.4763,E1 25.042,E2 884.5405} C_DIS
LIN {X 33.6228,Y -116.0576,Z 135,A -76.8835,B 24.9588,C -1.4828,E1 25.0461,E2 883.0254} C_DIS
LIN {X 37.5112,Y -114.8613,Z 135,A -74.9328,B 24.9586,C -1.4861,E1 25.0513,E2 881.0704} C_DIS
LIN {X 40.7019,Y -113.768,Z 135,A -73.4716,B 24.9589,C -1.4816,E1 25.0551,E2 879.623} C_DIS
LIN {X 43.4781,Y -112.7363,Z 135,A -71.9069,B 24.9583,C -1.4913,E1 25.0592,E2 878.0387} C_DIS
LIN {X 47.6001,Y -111.0589,Z 135,A -69.9739,B 24.9586,C -1.4858,E1 25.0642,E2 876.1232} C_DIS
LIN {X 50.6493,Y -109.7012,Z 135,A -68.3952,B 24.9586,C -1.4881,E1 25.0682,E2 874.543} C_DIS
LIN {X 52.9235,Y -108.6239,Z 135,A -67.226,B 24.9585,C -1.4888,E1 25.0711,E2 873.3751} C_DIS
LIN {X 55.6442,Y -107.2556,Z 135,A -65.6868,B 24.9581,C -1.4959,E1 25.075,E2 871.8234} C_DIS
LIN {X 58.6186,Y -105.6599,Z 135,A -64.1659,B 24.9581,C -1.4949,E1 25.0787,E2 870.3094} C_DIS
LIN {X 61.1712,Y -104.2028,Z 135,A -62.7702,B 24.958,C -1.4975,E1 25.0821,E2 868.9116} C_DIS
LIN {X 64.2991,Y -102.3026,Z 135,A -60.8771,B 24.9574,C -1.5086,E1 25.0866,E2 866.9983} C_DIS
LIN {X 67.4665,Y -100.2423,Z 135,A -59.2715,B 24.9577,C -1.5031,E1 25.0903,E2 865.4112} C_DIS
LIN {X 69.9001,Y -98.5607,Z 135,A -57.864,B 24.9575,C -1.5062,E1 25.0935,E2 864.0011} C_DIS
LIN {X 72.3183,Y -96.8,Z 135,A -56.3974,B 24.9572,C -1.5116,E1 25.0968,E2 862.527} C_DIS
LIN {X 75.5003,Y -94.3395,Z 135,A -54.5172,B 24.957,C -1.5145,E1 25.101,E2 860.647} C_DIS
LIN {X 78.3497,Y -91.9862,Z 135,A -52.7063,B 24.9566,C -1.5214,E1 25.1048,E2 858.8268} C_DIS
LIN {X 81.2745,Y -89.4125,Z 135,A -50.8573,B 24.9564,C -1.5258,E1 25.1087,E2 856.9747} C_DIS
LIN {X 84.3832,Y -86.4853,Z 135,A -48.8081,B 24.956,C -1.5319,E1 25.1128,E2 854.9195} C_DIS
LIN {X 87.4975,Y -83.3329,Z 135,A -46.8381,B 24.9561,C -1.5307,E1 25.1167,E2 852.9609} C_DIS
LIN {X 90.0022,Y -80.621,Z 135,A -45.0822,B 24.9558,C -1.5355,E1 25.12,E2 851.2015} C_DIS
LIN {X 92.4543,Y -77.797,Z 135,A -43.26,B 24.9554,C -1.5426,E1 25.1233,E2 849.3707} C_DIS
LIN {X 94.7909,Y -74.9331,Z 135,A -41.4629,B 24.955,C -1.5496,E1 25.1264,E2 847.5656} C_DIS
LIN {X 97.0379,Y -71.9987,Z 135,A -39.8744,B 24.9552,C -1.5462,E1 25.1291,E2 845.9926} C_DIS
LIN {X 98.7897,Y -69.5754,Z 135,A -38.4724,B 24.955,C -1.5494,E1 25.1313,E2 844.5899} C_DIS
LIN {X 100.4648,Y -67.1338,Z 135,A -37.0795,B 24.9548,C -1.5529,E1 25.1335,E2 843.1957} C_DIS
LIN {X 102.418,Y -64.1155,Z 135,A -35.2329,B 24.9541,C -1.5649,E1 25.1363,E2 841.3302} C_DIS
LIN {X 104.3955,Y -60.8428,Z 135,A -33.5822,B 24.9543,C -1.5621,E1 25.1387,E2 839.6945} C_DIS
LIN {X 105.8548,Y -58.2665,Z 135,A -32.0541,B 24.9537,C -1.5725,E1 25.1408,E2 838.1499} C_DIS
LIN {X 107.4511,Y -55.2648,Z 135,A -30.5933,B 24.9538,C -1.5698,E1 25.1426,E2 836.7032} C_DIS
LIN {X 109.022,Y -52.095,Z 135,A -28.837,B 24.9533,C -1.5788,E1 25.1448,E2 834.9349} C_DIS
LIN {X 110.623,Y -48.6081,Z 135,A -27.1192,B 24.9533,C -1.5793,E1 25.1467,E2 833.2253} C_DIS
LIN {X 112.0243,Y -45.2798,Z 135,A -25.2738,B 24.9525,C -1.5914,E1 25.1487,E2 831.3616} C_DIS
LIN {X 113.4028,Y -41.7137,Z 135,A -23.4201,B 24.9521,C -1.5991,E1 25.1506,E2 829.5} C_DIS
LIN {X 114.3904,Y -38.9234,Z 135,A -22.2137,B 24.9524,C -1.5936,E1 25.1516,E2 828.3133} C_DIS
LIN {X 115.5101,Y -35.4563,Z 135,A -20.3728,B 24.9517,C -1.6049,E1 25.1532,E2 826.4564} C_DIS
LIN {X 116.5639,Y -31.8296,Z 135,A -18.7161,B 24.9518,C -1.6039,E1 25.1544,E2 824.8115} C_DIS
LIN {X 117.4618,Y -28.3277,Z 135,A -17.2656,B 24.9523,C -1.5962,E1 25.1554,E2 823.3875} C_DIS
LIN {X 118.0636,Y -25.7058,Z 135,A -15.8783,B 24.9517,C -1.6059,E1 25.1563,E2 821.9852} C_DIS
LIN {X 118.5862,Y -23.1804,Z 135,A -14.5307,B 24.9511,C -1.6162,E1 25.157,E2 820.6214} C_DIS
LIN {X 119.1238,Y -20.2341,Z 135,A -13.289,B 24.9513,C -1.6119,E1 25.1576,E2 819.3971} C_DIS
LIN {X 119.5799,Y -17.3341,Z 135,A -11.742,B 24.9506,C -1.6242,E1 25.1583,E2 817.8302} C_DIS
LIN {X 119.9901,Y -14.2188,Z 135,A -10.3104,B 24.9504,C -1.6262,E1 25.1588,E2 816.4024} C_DIS
LIN {X 120.338,Y -10.9076,Z 135,A -8.5668,B 24.9496,C -1.6396,E1 25.1593,E2 814.6375} C_DIS
LIN {X 120.6113,Y -7.2624,Z 135,A -6.9419,B 24.9496,C -1.6399,E1 25.1596,E2 813.0215} C_DIS
LIN {X 120.7644,Y -4.0286,Z 135,A -5.2669,B 24.9489,C -1.6519,E1 25.1597,E2 811.3281} C_DIS
LIN {X 120.8331,Y 0,Z 135,A -3.3745,B 24.9485,C -1.6573,E1 25.1597,E2 809.4344} C_DIS
LIN {X 120.7644,Y 4.0286,Z 135,A -1.5156,B 24.9483,C -1.6609,E1 25.1597,E2 807.5779} C_DIS
LIN {X 120.602,Y 7.4139,Z 135,A 0.0007,B 24.9483,C -1.6617,E1 25.1594,E2 806.0689} C_DIS
LIN {X 120.3496,Y 10.7772,Z 135,A 1.6001,B 24.9479,C -1.6668,E1 25.159,E2 804.4667} C_DIS
LIN {X 120.0489,Y 13.7259,Z 135,A 3.085,B 24.9474,C -1.6754,E1 25.1586,E2 802.9705} C_DIS
LIN {X 119.5215,Y 17.743,Z 135,A 4.8581,B 24.9474,C -1.6741,E1 25.1579,E2 801.2108} C_DIS
LIN {X 119.0557,Y 20.6381,Z 135,A 6.2195,B 24.9473,C -1.6771,E1 25.1573,E2 799.8503} C_DIS
LIN {X 118.5203,Y 23.517,Z 135,A 7.5929,B 24.9471,C -1.6808,E1 25.1565,E2 798.4763} C_DIS
LIN {X 117.9216,Y 26.3545,Z 135,A 9.1089,B 24.9463,C -1.6922,E1 25.1556,E2 796.9422} C_DIS
Enddeposition()
END
